KUKA KRL program: MyProgram_192().src

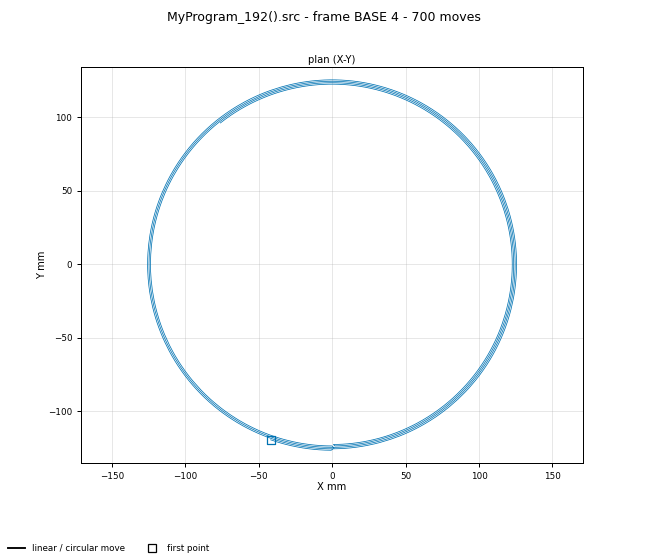
[picture p0: tool path of MyProgram_192().src in frame BASE 4, 700 of 700 moves have a stored position in this frame; points joined in program order, loops and branches not executed]
&ACCESS RVP
&REL 1
&PARAM TEMPLATE = C:\KRC\Roboter\Template\vorgabe
&PARAM EDITMASK = *
DEF MyProgram_192()
; ---- Setting reference (Base) ----
$BASE = BASE_DATA[4]

; --------------------------
; ---- Setting tool (TCP) ----
$TOOL = TOOL_DATA[3]
; --------------------------

$VEL.CP = VEL_APROX_PRINT
Startdeposition()
$VEL.CP = VEL_PRINT
LIN {X -41.8046,Y -119.4809,Z 139,A -112.1898,B 24.9633,C -1.4001,E1 24.9485,E2 558.5305} C_DIS
LIN {X -38.0832,Y -120.719,Z 139,A -110.4755,B 24.9635,C -1.3957,E1 24.953,E2 556.8235} C_DIS
LIN {X -35.043,Y -121.6367,Z 139,A -109.0218,B 24.9635,C -1.3954,E1 24.9569,E2 555.368} C_DIS
LIN {X -31.8921,Y -122.5017,Z 139,A -107.3287,B 24.963,C -1.405,E1 24.9616,E2 553.6497} C_DIS
LIN {X -27.5144,Y -123.5583,Z 139,A -105.3425,B 24.9632,C -1.4014,E1 24.967,E2 551.6695} C_DIS
LIN {X -23.703,Y -124.3439,Z 139,A -103.7035,B 24.9636,C -1.3947,E1 24.9714,E2 550.0445} C_DIS
LIN {X -20.2277,Y -124.9578,Z 139,A -102.0069,B 24.9633,C -1.399,E1 24.9761,E2 548.336} C_DIS
LIN {X -16.3797,Y -125.5188,Z 139,A -100.3777,B 24.9637,C -1.3922,E1 24.9806,E2 546.7217} C_DIS
LIN {X -12.7728,Y -125.9388,Z 139,A -98.5892,B 24.9633,C -1.3991,E1 24.9856,E2 544.9157} C_DIS
LIN {X -8.9623,Y -126.2657,Z 139,A -96.8687,B 24.9633,C -1.3986,E1 24.9904,E2 543.1957} C_DIS
LIN {X -4.8152,Y -126.4916,Z 139,A -95.0556,B 24.9635,C -1.3954,E1 24.9954,E2 541.3897} C_DIS
LIN {X -0.6506,Y -126.5815,Z 139,A -93.2386,B 24.9637,C -1.3924,E1 25.0005,E2 539.5799} C_DIS
LIN {X -0.6506,Y -126.5815,Z 139,A -93.2386,B 24.9637,C -1.3924,E1 25.0005,E2 539.5799} C_DIS
Enddeposition()
LIN {X 0.8997,Y -125.5994,Z 139,A -93.1322,B 24.9643,C -1.3803,E1 25.0007,E2 539.5021} C_DIS
Startdeposition()
$VEL.CP = VEL_PRINT
LIN {X -2.5774,Y -125.5787,Z 139,A -94.9255,B 24.9649,C -1.3699,E1 24.9956,E2 541.3201} C_DIS
LIN {X -6.6331,Y -125.4293,Z 139,A -96.7717,B 24.9649,C -1.3699,E1 24.9905,E2 543.1665} C_DIS
LIN {X -10.6993,Y -125.1476,Z 139,A -98.5659,B 24.9647,C -1.3732,E1 24.9855,E2 544.9538} C_DIS
LIN {X -14.9192,Y -124.7148,Z 139,A -100.4884,B 24.9647,C -1.374,E1 24.9802,E2 546.8756} C_DIS
LIN {X -18.8934,Y -124.1753,Z 139,A -102.3022,B 24.9646,C -1.3752,E1 24.9752,E2 548.688} C_DIS
LIN {X -22.2036,Y -123.6258,Z 139,A -103.8436,B 24.9646,C -1.3752,E1 24.9709,E2 550.2309} C_DIS
LIN {X -25.9892,Y -122.8868,Z 139,A -105.6556,B 24.9646,C -1.3734,E1 24.9659,E2 552.0493} C_DIS
LIN {X -28.9108,Y -122.2325,Z 139,A -107.185,B 24.965,C -1.3663,E1 24.9617,E2 553.5976} C_DIS
LIN {X -33.6478,Y -121.0131,Z 139,A -109.19,B 24.9644,C -1.3785,E1 24.9564,E2 555.5766} C_DIS
LIN {X -36.8186,Y -120.0862,Z 139,A -110.6976,B 24.9644,C -1.3796,E1 24.9523,E2 557.0842} C_DIS
LIN {X -39.7861,Y -119.1359,Z 139,A -112.2561,B 24.9646,C -1.3742,E1 24.9482,E2 558.6584} C_DIS
LIN {X -43.8401,Y -117.7047,Z 139,A -114.0437,B 24.9641,C -1.3842,E1 24.9435,E2 560.4258} C_DIS
LIN {X -46.4102,Y -116.7164,Z 139,A -115.4613,B 24.9644,C -1.3778,E1 24.9398,E2 561.8618} C_DIS
LIN {X -50.5279,Y -114.9946,Z 139,A -117.4765,B 24.9643,C -1.3809,E1 24.9346,E2 563.8741} C_DIS
LIN {X -53.8675,Y -113.4665,Z 139,A -119.0475,B 24.9639,C -1.3878,E1 24.9307,E2 565.4326} C_DIS
LIN {X -57.4932,Y -111.6742,Z 139,A -120.8939,B 24.9639,C -1.3901,E1 24.9261,E2 567.2786} C_DIS
LIN {X -60.8547,Y -109.8792,Z 139,A -122.6643,B 24.9638,C -1.391,E1 24.9217,E2 569.0519} C_DIS
LIN {X -64.9208,Y -107.5265,Z 139,A -125.2363,B 24.9646,C -1.3741,E1 24.9154,E2 571.6717} C_DIS
LIN {X -68.1564,Y -105.506,Z 139,A -126.6649,B 24.9637,C -1.3913,E1 24.9122,E2 573.0641} C_DIS
LIN {X -71.0171,Y -103.6017,Z 139,A -128.2398,B 24.9637,C -1.3936,E1 24.9085,E2 574.6388} C_DIS
LIN {X -74.697,Y -100.9815,Z 139,A -130.2962,B 24.9634,C -1.3974,E1 24.9039,E2 576.6934} C_DIS
LIN {X -77.4345,Y -98.8973,Z 139,A -132.2032,B 24.9641,C -1.3847,E1 24.8996,E2 578.6376} C_DIS
LIN {X -80.408,Y -96.4958,Z 139,A -133.6399,B 24.9632,C -1.4021,E1 24.8966,E2 580.0383} C_DIS
LIN {X -83.6363,Y -93.711,Z 139,A -135.5875,B 24.963,C -1.4059,E1 24.8925,E2 581.9846} C_DIS
LIN {X -86.9695,Y -90.6262,Z 139,A -137.6592,B 24.9627,C -1.4102,E1 24.8883,E2 584.0545} C_DIS
LIN {X -90.0345,Y -87.582,Z 139,A -139.6608,B 24.9626,C -1.4131,E1 24.8843,E2 586.0578} C_DIS
LIN {X -92.6006,Y -84.864,Z 139,A -141.6419,B 24.9631,C -1.4044,E1 24.8805,E2 588.0684} C_DIS
LIN {X -95.0006,Y -82.1687,Z 139,A -143.0168,B 24.9622,C -1.4205,E1 24.8781,E2 589.411} C_DIS
LIN {X -97.863,Y -78.7375,Z 139,A -144.9662,B 24.9617,C -1.4295,E1 24.8746,E2 591.3482} C_DIS
LIN {X -100.4945,Y -75.3509,Z 139,A -147.0461,B 24.9617,C -1.4287,E1 24.8711,E2 593.4399} C_DIS
LIN {X -102.9709,Y -71.929,Z 139,A -149.1222,B 24.9619,C -1.4269,E1 24.8677,E2 595.5306} C_DIS
LIN {X -105.0542,Y -68.8508,Z 139,A -150.9071,B 24.9619,C -1.4272,E1 24.865,E2 597.3235} C_DIS
LIN {X -106.8737,Y -65.9915,Z 139,A -152.244,B 24.9611,C -1.4408,E1 24.863,E2 598.6349} C_DIS
LIN {X -109.1521,Y -62.1496,Z 139,A -154.2487,B 24.9607,C -1.4478,E1 24.8602,E2 600.6332} C_DIS
LIN {X -110.9704,Y -58.8396,Z 139,A -155.9668,B 24.9605,C -1.4529,E1 24.858,E2 602.3485} C_DIS
LIN {X -113.9832,Y -52.7646,Z 139,A -159.0137,B 24.9599,C -1.4638,E1 24.8543,E2 605.3858} C_DIS
LIN {X -115.3845,Y -49.626,Z 139,A -160.6837,B 24.9599,C -1.4638,E1 24.8524,E2 607.065} C_DIS
LIN {X -116.9285,Y -45.8711,Z 139,A -162.312,B 24.959,C -1.4793,E1 24.8507,E2 608.6654} C_DIS
LIN {X -118.071,Y -42.844,Z 139,A -163.9544,B 24.9592,C -1.4763,E1 24.8491,E2 610.3244} C_DIS
LIN {X -119.1423,Y -39.7671,Z 139,A -165.4335,B 24.9589,C -1.4811,E1 24.8477,E2 611.8003} C_DIS
LIN {X -120.1236,Y -36.6965,Z 139,A -166.9045,B 24.9587,C -1.4856,E1 24.8465,E2 613.2691} C_DIS
LIN {X -121.1356,Y -33.2072,Z 139,A -168.7783,B 24.9589,C -1.481,E1 24.8451,E2 615.1646} C_DIS
LIN {X -122.133,Y -29.3235,Z 139,A -170.7253,B 24.9589,C -1.4815,E1 24.8438,E2 617.1219} C_DIS
LIN {X -123.4003,Y -23.4251,Z 139,A -172.8757,B 24.9569,C -1.5171,E1 24.8426,E2 619.2} C_DIS
LIN {X -124.2205,Y -18.6016,Z 139,A -175.544,B 24.9576,C -1.5047,E1 24.8414,E2 621.9139} C_DIS
LIN {X -124.7295,Y -14.7961,Z 139,A -177.2038,B 24.957,C -1.5145,E1 24.8408,E2 623.5604} C_DIS
LIN {X -125.2275,Y -9.7372,Z 139,A -179.7895,B 24.9573,C -1.5101,E1 24.8401,E2 626.1719} C_DIS
LIN {X -125.5171,Y -4.6805,Z 139,A 178.1039,B 24.9563,C -1.5267,E1 24.8399,E2 628.2515} C_DIS
LIN {X -125.5893,Y -1.9388,Z 139,A 176.6889,B 24.9565,C -1.5236,E1 24.8398,E2 629.6827} C_DIS
LIN {X -125.5414,Y 4.0033,Z 139,A 174.0819,B 24.9557,C -1.537,E1 24.8399,E2 632.2733} C_DIS
LIN {X -125.3591,Y 7.8425,Z 139,A 172.3326,B 24.9554,C -1.543,E1 24.8402,E2 634.0188} C_DIS
LIN {X -124.8359,Y 13.8763,Z 139,A 169.6269,B 24.9547,C -1.5546,E1 24.8409,E2 636.7132} C_DIS
LIN {X -124.0149,Y 19.9294,Z 139,A 166.6755,B 24.9547,C -1.5564,E1 24.8421,E2 639.6779} C_DIS
LIN {X -123.367,Y 23.5991,Z 139,A 165.0734,B 24.954,C -1.5663,E1 24.8429,E2 641.2658} C_DIS
LIN {X -122.5721,Y 27.4356,Z 139,A 163.0882,B 24.9542,C -1.5633,E1 24.844,E2 643.2698} C_DIS
LIN {X -121.449,Y 32.0403,Z 139,A 161.0453,B 24.9535,C -1.5756,E1 24.8454,E2 645.2954} C_DIS
LIN {X -120.3646,Y 35.9036,Z 139,A 159.278,B 24.953,C -1.5843,E1 24.8468,E2 647.0523} C_DIS
LIN {X -119.2699,Y 39.3837,Z 139,A 157.5521,B 24.9528,C -1.5868,E1 24.8483,E2 648.7819} C_DIS
LIN {X -118.0874,Y 42.7983,Z 139,A 155.8874,B 24.9526,C -1.5913,E1 24.8498,E2 650.4453} C_DIS
LIN {X -117.06,Y 45.5329,Z 139,A 154.2556,B 24.9531,C -1.5822,E1 24.8515,E2 652.108} C_DIS
LIN {X -115.836,Y 48.5627,Z 139,A 153.0432,B 24.9521,C -1.5992,E1 24.8527,E2 653.2867} C_DIS
LIN {X -113.2763,Y 54.2656,Z 139,A 150.184,B 24.9516,C -1.6076,E1 24.8561,E2 656.1415} C_DIS
LIN {X -111.744,Y 57.356,Z 139,A 148.3559,B 24.952,C -1.601,E1 24.8584,E2 657.9951} C_DIS
LIN {X -109.8749,Y 60.8626,Z 139,A 146.0208,B 24.953,C -1.5833,E1 24.8617,E2 660.3848} C_DIS
LIN {X -107.1204,Y 65.5894,Z 139,A 144.2085,B 24.9508,C -1.6208,E1 24.8641,E2 662.117} C_DIS
LIN {X -104.7423,Y 69.3244,Z 139,A 142.1709,B 24.9505,C -1.6258,E1 24.8672,E2 664.153} C_DIS
LIN {X -102.4969,Y 72.603,Z 139,A 140.3858,B 24.9501,C -1.6321,E1 24.8701,E2 665.9319} C_DIS
LIN {X -100.006,Y 75.9979,Z 139,A 138.3651,B 24.9501,C -1.6329,E1 24.8735,E2 667.9603} C_DIS
LIN {X -97.3017,Y 79.43,Z 139,A 136.4034,B 24.9496,C -1.6397,E1 24.8769,E2 669.9151} C_DIS
LIN {X -94.3922,Y 82.8673,Z 139,A 134.2991,B 24.9494,C -1.6428,E1 24.8807,E2 672.0215} C_DIS
LIN {X -91.6174,Y 85.9251,Z 139,A 132.405,B 24.9492,C -1.6471,E1 24.8843,E2 673.9137} C_DIS
LIN {X -88.5694,Y 89.0629,Z 139,A 130.4421,B 24.9488,C -1.6535,E1 24.8881,E2 675.8697} C_DIS
LIN {X -85.3469,Y 92.1562,Z 139,A 128.3653,B 24.9486,C -1.6566,E1 24.8924,E2 677.9476} C_DIS
LIN {X -82.2121,Y 94.9632,Z 139,A 126.4267,B 24.9483,C -1.6602,E1 24.8964,E2 679.8854} C_DIS
LIN {X -78.6759,Y 97.9126,Z 139,A 124.372,B 24.9479,C -1.667,E1 24.9008,E2 681.9317} C_DIS
LIN {X -75.5113,Y 100.3734,Z 139,A 122.5578,B 24.9476,C -1.6716,E1 24.9048,E2 683.7416} C_DIS
LIN {X -72.0749,Y 102.8694,Z 139,A 120.5324,B 24.9476,C -1.6716,E1 24.9095,E2 685.774} C_DIS
LIN {X -68.4195,Y 105.3352,Z 139,A 118.5413,B 24.9473,C -1.6765,E1 24.9141,E2 687.7599} C_DIS
LIN {X -64.6224,Y 107.7071,Z 139,A 115.7068,B 24.9493,C -1.6444,E1 24.9211,E2 690.6795} C_DIS
LIN {X -59.4468,Y 110.6473,Z 139,A 113.7306,B 24.9469,C -1.6827,E1 24.9257,E2 692.5704} C_DIS
LIN {X -55.8231,Y 112.5172,Z 139,A 112.2269,B 24.9457,C -1.7022,E1 24.9293,E2 694.0317} C_DIS
LIN {X -52.1716,Y 114.2574,Z 139,A 109.967,B 24.9467,C -1.6859,E1 24.9352,E2 696.3359} C_DIS
LIN {X -48.6833,Y 115.7856,Z 139,A 108.4077,B 24.9461,C -1.6967,E1 24.9391,E2 697.8732} C_DIS
LIN {X -45.6353,Y 117.0202,Z 139,A 106.8995,B 24.9459,C -1.6984,E1 24.943,E2 699.3806} C_DIS
LIN {X -41.9744,Y 118.3845,Z 139,A 103.8529,B 24.9494,C -1.6428,E1 24.9515,E2 702.5654} C_DIS
LIN {X -34.5296,Y 120.7665,Z 139,A 100.6379,B 24.9482,C -1.6627,E1 24.9599,E2 705.7385} C_DIS
LIN {X -28.6672,Y 122.2908,Z 139,A 98.159,B 24.9472,C -1.6783,E1 24.9666,E2 708.1834} C_DIS
LIN {X -24.1576,Y 123.2602,Z 139,A 96.5853,B 24.9455,C -1.7048,E1 24.9707,E2 709.6962} C_DIS
LIN {X -20.4182,Y 123.9335,Z 139,A 94.906,B 24.9453,C -1.7086,E1 24.9753,E2 711.3681} C_DIS
LIN {X -16.5856,Y 124.5044,Z 139,A 93.1652,B 24.9451,C -1.711,E1 24.9801,E2 713.1045} C_DIS
LIN {X -13.4064,Y 124.8865,Z 139,A 91.6264,B 24.9453,C -1.7082,E1 24.9844,E2 714.651} C_DIS
LIN {X -9.281,Y 125.2608,Z 139,A 89.7847,B 24.9451,C -1.7113,E1 24.9895,E2 716.4861} C_DIS
LIN {X -5.3106,Y 125.4925,Z 139,A 87.933,B 24.9451,C -1.7102,E1 24.9947,E2 718.3411} C_DIS
LIN {X -1.4943,Y 125.5967,Z 139,A 86.1631,B 24.9452,C -1.7093,E1 24.9996,E2 720.1132} C_DIS
LIN {X 2.1011,Y 125.5866,Z 139,A 84.5803,B 24.9451,C -1.7123,E1 25.004,E2 721.6887} C_DIS
LIN {X 6.1932,Y 125.4514,Z 139,A 82.7367,B 24.945,C -1.7136,E1 25.0092,E2 723.5288} C_DIS
LIN {X 9.8797,Y 125.2168,Z 139,A 80.918,B 24.9454,C -1.7071,E1 25.0143,E2 725.362} C_DIS
LIN {X 13.9908,Y 124.8236,Z 139,A 79.0735,B 24.9453,C -1.7087,E1 25.0194,E2 727.2014} C_DIS
LIN {X 17.7134,Y 124.3487,Z 139,A 77.4381,B 24.9451,C -1.712,E1 25.0239,E2 728.8277} C_DIS
LIN {X 21.5145,Y 123.7492,Z 139,A 75.65,B 24.9452,C -1.7098,E1 25.0288,E2 730.6192} C_DIS
LIN {X 25.5833,Y 122.9721,Z 139,A 73.4688,B 24.9462,C -1.6949,E1 25.0349,E2 732.8329} C_DIS
LIN {X 28.8679,Y 122.2428,Z 139,A 72.1891,B 24.9454,C -1.7063,E1 25.0383,E2 734.0838} C_DIS
LIN {X 32.3878,Y 121.3563,Z 139,A 70.5867,B 24.9454,C -1.7079,E1 25.0426,E2 735.6801} C_DIS
LIN {X 36.3536,Y 120.2285,Z 139,A 68.5283,B 24.946,C -1.6979,E1 25.0482,E2 737.7586} C_DIS
LIN {X 40.896,Y 118.7598,Z 139,A 66.5494,B 24.9455,C -1.7057,E1 25.0533,E2 739.7152} C_DIS
LIN {X 45.1754,Y 117.199,Z 139,A 64.4528,B 24.9457,C -1.7028,E1 25.0588,E2 741.8142} C_DIS
LIN {X 48.4633,Y 115.8775,Z 139,A 62.9005,B 24.9456,C -1.7042,E1 25.0628,E2 743.3596} C_DIS
LIN {X 51.3868,Y 114.611,Z 139,A 61.4504,B 24.9456,C -1.7027,E1 25.0665,E2 744.8097} C_DIS
LIN {X 54.4859,Y 113.1711,Z 139,A 59.5276,B 24.9469,C -1.683,E1 25.0715,E2 746.7742} C_DIS
LIN {X 57.6312,Y 111.6038,Z 139,A 58.3046,B 24.9459,C -1.6995,E1 25.0744,E2 747.9549} C_DIS
LIN {X 60.2766,Y 110.1975,Z 139,A 56.2801,B 24.948,C -1.6653,E1 25.0796,E2 750.0543} C_DIS
LIN {X 64.4594,Y 107.8042,Z 139,A 54.6424,B 24.9465,C -1.6895,E1 25.0834,E2 751.6298} C_DIS
LIN {X 68.1071,Y 105.5381,Z 139,A 52.6395,B 24.9468,C -1.6842,E1 25.0881,E2 753.6387} C_DIS
LIN {X 71.9524,Y 102.9547,Z 139,A 50.5794,B 24.9469,C -1.6833,E1 25.0928,E2 755.694} C_DIS
LIN {X 75.4343,Y 100.4315,Z 139,A 48.6447,B 24.947,C -1.6811,E1 25.0972,E2 757.627} C_DIS
LIN {X 79.735,Y 97.0517,Z 139,A 46.049,B 24.9477,C -1.6714,E1 25.1029,E2 760.2359} C_DIS
LIN {X 83.6029,Y 93.7409,Z 139,A 43.8076,B 24.9477,C -1.6707,E1 25.1076,E2 762.47} C_DIS
LIN {X 86.9996,Y 90.5972,Z 139,A 41.7098,B 24.9479,C -1.667,E1 25.1118,E2 764.5681} C_DIS
LIN {X 90.044,Y 87.5722,Z 139,A 39.7496,B 24.9482,C -1.6625,E1 25.1157,E2 766.5303} C_DIS
LIN {X 92.3902,Y 85.0928,Z 139,A 38.3722,B 24.9479,C -1.6681,E1 25.1183,E2 767.8887} C_DIS
LIN {X 94.875,Y 82.314,Z 139,A 36.5164,B 24.9486,C -1.6563,E1 25.1217,E2 769.764} C_DIS
LIN {X 97.6304,Y 79.0258,Z 139,A 34.5782,B 24.9488,C -1.6525,E1 25.1252,E2 771.7022} C_DIS
LIN {X 100.3697,Y 75.5162,Z 139,A 32.5251,B 24.9492,C -1.6463,E1 25.1287,E2 773.7601} C_DIS
LIN {X 102.808,Y 72.1619,Z 139,A 30.6579,B 24.9494,C -1.6427,E1 25.1317,E2 775.6267} C_DIS
LIN {X 105.2436,Y 68.5606,Z 139,A 28.7003,B 24.9497,C -1.6388,E1 25.1347,E2 777.5837} C_DIS
LIN {X 107.643,Y 64.7288,Z 139,A 26.9349,B 24.9491,C -1.6484,E1 25.1373,E2 779.3177} C_DIS
LIN {X 109.422,Y 61.6733,Z 139,A 25.0482,B 24.9502,C -1.63,E1 25.1399,E2 781.2379} C_DIS
LIN {X 111.6062,Y 57.6225,Z 139,A 22.4385,B 24.9521,C -1.5982,E1 25.1434,E2 783.9088} C_DIS
LIN {X 113.7419,Y 53.2865,Z 139,A 20.7741,B 24.9509,C -1.6193,E1 25.1453,E2 785.5145} C_DIS
LIN {X 115.2836,Y 49.8595,Z 139,A 19.1857,B 24.9508,C -1.6207,E1 25.1471,E2 787.0909} C_DIS
LIN {X 116.5335,Y 46.8639,Z 139,A 17.7529,B 24.9508,C -1.6188,E1 25.1486,E2 788.5204} C_DIS
LIN {X 117.6624,Y 43.9529,Z 139,A 16.2668,B 24.9513,C -1.6114,E1 25.1501,E2 790.0158} C_DIS
LIN {X 119.789,Y 37.7772,Z 139,A 13.5675,B 24.951,C -1.6167,E1 25.1525,E2 792.6873} C_DIS
LIN {X 121.2092,Y 32.9393,Z 139,A 10.9939,B 24.9523,C -1.5954,E1 25.1545,E2 795.2963} C_DIS
LIN {X 122.115,Y 29.398,Z 139,A 9.039,B 24.9535,C -1.5754,E1 25.1558,E2 797.2871} C_DIS
LIN {X 122.8724,Y 26.0559,Z 139,A 7.7703,B 24.9529,C -1.5855,E1 25.1566,E2 798.5245} C_DIS
LIN {X 123.6152,Y 22.2629,Z 139,A 6.0298,B 24.9532,C -1.5811,E1 25.1575,E2 800.2653} C_DIS
LIN {X 124.2666,Y 18.2882,Z 139,A 4.1797,B 24.9536,C -1.5745,E1 25.1583,E2 802.12} C_DIS
LIN {X 124.7327,Y 14.7691,Z 139,A 2.6323,B 24.9536,C -1.573,E1 25.1588,E2 803.6619} C_DIS
LIN {X 125.1456,Y 10.7228,Z 139,A 0.7912,B 24.954,C -1.5677,E1 25.1593,E2 805.5045} C_DIS
LIN {X 125.4112,Y 6.9924,Z 139,A -1.0044,B 24.9546,C -1.5574,E1 25.1596,E2 807.3136} C_DIS
LIN {X 125.5653,Y 3.1414,Z 139,A -2.6651,B 24.9546,C -1.5567,E1 25.1598,E2 808.9662} C_DIS
LIN {X 125.6025,Y -0.7041,Z 139,A -4.4232,B 24.9549,C -1.5508,E1 25.1598,E2 810.7279} C_DIS
LIN {X 125.5084,Y -4.9039,Z 139,A -6.3178,B 24.9552,C -1.5456,E1 25.1596,E2 812.6234} C_DIS
LIN {X 125.28,Y -9.018,Z 139,A -8.197,B 24.9556,C -1.5394,E1 25.1593,E2 814.5059} C_DIS
LIN {X 124.9403,Y -12.9066,Z 139,A -9.9541,B 24.9559,C -1.5347,E1 25.1588,E2 816.2637} C_DIS
LIN {X 124.5518,Y -16.2243,Z 139,A -11.4431,B 24.9561,C -1.5315,E1 25.1583,E2 817.7514} C_DIS
LIN {X 123.9986,Y -20.0282,Z 139,A -13.2581,B 24.9566,C -1.5226,E1 25.1575,E2 819.5769} C_DIS
LIN {X 123.4086,Y -23.3815,Z 139,A -14.6965,B 24.9566,C -1.5234,E1 25.1568,E2 821.0049} C_DIS
LIN {X 121.8269,Y -30.5719,Z 139,A -18.0743,B 24.9572,C -1.5115,E1 25.1547,E2 824.3912} C_DIS
LIN {X 120.8473,Y -34.2409,Z 139,A -20.0519,B 24.9582,C -1.4932,E1 25.1532,E2 826.4005} C_DIS
LIN {X 119.3517,Y -39.1383,Z 139,A -22.0859,B 24.9578,C -1.5013,E1 25.1516,E2 828.4039} C_DIS
LIN {X 117.7927,Y -43.605,Z 139,A -24.2456,B 24.9582,C -1.4943,E1 25.1495,E2 830.5679} C_DIS
LIN {X 116.5292,Y -46.8746,Z 139,A -26.2206,B 24.9595,C -1.47,E1 25.1474,E2 832.5893} C_DIS
LIN {X 115.1052,Y -50.2722,Z 139,A -27.5204,B 24.9587,C -1.4843,E1 25.1461,E2 833.8482} C_DIS
LIN {X 113.3225,Y -54.1691,Z 139,A -29.5136,B 24.9592,C -1.4763,E1 25.1437,E2 835.8495} C_DIS
LIN {X 111.3795,Y -58.0604,Z 139,A -31.4306,B 24.9593,C -1.4738,E1 25.1413,E2 837.7624} C_DIS
LIN {X 109.7344,Y -61.1163,Z 139,A -33.049,B 24.9597,C -1.4672,E1 25.1391,E2 839.3878} C_DIS
LIN {X 107.6373,Y -64.7383,Z 139,A -34.9579,B 24.96,C -1.4616,E1 25.1364,E2 841.3001} C_DIS
LIN {X 105.4653,Y -68.2191,Z 139,A -36.8491,B 24.9603,C -1.4551,E1 25.1335,E2 843.197} C_DIS
LIN {X 103.1553,Y -71.6641,Z 139,A -38.7026,B 24.9605,C -1.4517,E1 25.1306,E2 845.0494} C_DIS
LIN {X 100.6382,Y -75.1579,Z 139,A -41.1904,B 24.9623,C -1.4195,E1 25.1264,E2 847.6011} C_DIS
LIN {X 97.7463,Y -78.8822,Z 139,A -42.5715,B 24.9605,C -1.453,E1 25.1241,E2 848.8969} C_DIS
LIN {X 93.386,Y -83.9992,Z 139,A -46.2121,B 24.9625,C -1.4156,E1 25.1173,E2 852.6094} C_DIS
LIN {X 90.744,Y -86.8461,Z 139,A -47.7215,B 24.962,C -1.4244,E1 25.1145,E2 854.0913} C_DIS
LIN {X 85.6075,Y -91.9135,Z 139,A -50.8034,B 24.9619,C -1.427,E1 25.1083,E2 857.1543} C_DIS
LIN {X 80.0109,Y -96.8246,Z 139,A -54.0155,B 24.9618,C -1.4284,E1 25.1016,E2 860.3503} C_DIS
LIN {X 76.5271,Y -99.6013,Z 139,A -56.3022,B 24.9627,C -1.411,E1 25.0965,E2 862.6698} C_DIS
LIN {X 73.5795,Y -101.7979,Z 139,A -58.311,B 24.9638,C -1.3907,E1 25.0919,E2 864.7194} C_DIS
LIN {X 70.45,Y -103.9877,Z 139,A -59.6437,B 24.9629,C -1.4077,E1 25.0889,E2 866.0072} C_DIS
LIN {X 66.86,Y -106.3321,Z 139,A -61.6238,B 24.9631,C -1.4027,E1 25.0842,E2 867.993} C_DIS
LIN {X 63.4602,Y -108.3954,Z 139,A -63.4037,B 24.9632,C -1.401,E1 25.08,E2 869.7714} C_DIS
LIN {X 59.7756,Y -110.4706,Z 139,A -65.4413,B 24.9637,C -1.392,E1 25.075,E2 871.8241} C_DIS
LIN {X 55.8397,Y -112.509,Z 139,A -67.2931,B 24.9634,C -1.3972,E1 25.0704,E2 873.6587} C_DIS
LIN {X 52.8798,Y -113.9299,Z 139,A -68.765,B 24.9634,C -1.3961,E1 25.0667,E2 875.1294} C_DIS
LIN {X 49.8421,Y -115.2911,Z 139,A -70.3195,B 24.9637,C -1.3919,E1 25.0627,E2 876.6899} C_DIS
LIN {X 46.2319,Y -116.788,Z 139,A -72.1209,B 24.9639,C -1.3884,E1 25.058,E2 878.4956} C_DIS
LIN {X 39.8318,Y -119.1208,Z 139,A -75.2446,B 24.9641,C -1.3835,E1 25.0498,E2 881.6245} C_DIS
LIN {X 32.398,Y -121.3536,Z 139,A -78.6786,B 24.9641,C -1.3847,E1 25.0406,E2 885.0497} C_DIS
LIN {X 29.093,Y -122.1886,Z 139,A -80.3728,B 24.9645,C -1.3762,E1 25.036,E2 886.7615} C_DIS
LIN {X 23.7626,Y -123.3358,Z 139,A -82.7302,B 24.9643,C -1.3804,E1 25.0296,E2 889.106} C_DIS
LIN {X 20.4803,Y -123.9231,Z 139,A -84.2751,B 24.9644,C -1.378,E1 25.0253,E2 890.6549} C_DIS
LIN {X 16.4838,Y -124.5178,Z 139,A -86.1039,B 24.9644,C -1.3774,E1 25.0202,E2 892.4835} C_DIS
LIN {X 13.0103,Y -124.9291,Z 139,A -87.7746,B 24.9647,C -1.3728,E1 25.0156,E2 894.1641} C_DIS
LIN {X 9.2051,Y -125.2663,Z 139,A -89.4526,B 24.9646,C -1.3751,E1 25.0109,E2 895.8357} C_DIS
LIN {X 5.1896,Y -125.4972,Z 139,A -91.3048,B 24.9646,C -1.3735,E1 25.0058,E2 897.691} C_DIS
LIN {X 1.4055,Y -125.5982,Z 139,A -93.1062,B 24.9649,C -1.3693,E1 25.0007,E2 899.5021} C_DIS
LIN {X 1.4055,Y -125.5982,Z 139,A -93.1062,B 24.9649,C -1.3693,E1 25.0007,E2 899.5021} C_DIS
Enddeposition()
LIN {X 0.8898,Y -124.6193,Z 139,A -92.6917,B 24.7402,C -1.3712,E1 24.7777,E2 899.052} C_DIS
Startdeposition()
$VEL.CP = VEL_PRINT
LIN {X 4.2848,Y -124.5527,Z 139,A -90.8344,B 24.7394,C -1.386,E1 24.783,E2 897.1598} C_DIS
LIN {X 8.4379,Y -124.3407,Z 139,A -88.8956,B 24.7394,C -1.3881,E1 24.7884,E2 895.2167} C_DIS
LIN {X 12.3432,Y -124.013,Z 139,A -87.1688,B 24.7394,C -1.3855,E1 24.7932,E2 893.4973} C_DIS
LIN {X 16.3271,Y -123.5509,Z 139,A -85.358,B 24.7394,C -1.385,E1 24.7982,E2 891.689} C_DIS
LIN {X 20.3865,Y -122.9462,Z 139,A -83.4647,B 24.7394,C -1.3867,E1 24.8035,E2 889.7935} C_DIS
LIN {X 24.246,Y -122.2451,Z 139,A -81.4769,B 24.7388,C -1.3973,E1 24.809,E2 887.7827} C_DIS
LIN {X 29.506,Y -121.082,Z 139,A -79.1186,B 24.739,C -1.3939,E1 24.8154,E2 885.436} C_DIS
LIN {X 35.6088,Y -119.4306,Z 139,A -76.0112,B 24.7383,C -1.407,E1 24.8238,E2 882.3023} C_DIS
LIN {X 38.7371,Y -118.4534,Z 139,A -74.8992,B 24.7393,C -1.3893,E1 24.8266,E2 881.2349} C_DIS
LIN {X 43.968,Y -116.6113,Z 139,A -72.2971,B 24.7389,C -1.3952,E1 24.8335,E2 878.624} C_DIS
LIN {X 46.6782,Y -115.5528,Z 139,A -70.9573,B 24.7389,C -1.3973,E1 24.837,E2 877.2824} C_DIS
LIN {X 49.9084,Y -114.1958,Z 139,A -69.3718,B 24.7388,C -1.3984,E1 24.841,E2 875.6979} C_DIS
LIN {X 52.4782,Y -113.037,Z 139,A -68.0984,B 24.7388,C -1.3993,E1 24.8442,E2 874.4255} C_DIS
LIN {X 55.3568,Y -111.6556,Z 139,A -66.5505,B 24.7384,C -1.4057,E1 24.8482,E2 872.8665} C_DIS
LIN {X 59.3234,Y -109.6022,Z 139,A -64.4739,B 24.7381,C -1.4104,E1 24.8533,E2 870.7847} C_DIS
LIN {X 62.8966,Y -107.5911,Z 139,A -62.6268,B 24.7381,C -1.412,E1 24.8578,E2 868.9394} C_DIS
LIN {X 66.2174,Y -105.58,Z 139,A -60.7849,B 24.7377,C -1.4183,E1 24.8622,E2 867.0885} C_DIS
LIN {X 72.0177,Y -101.7117,Z 139,A -57.8149,B 24.738,C -1.4129,E1 24.869,E2 864.1414} C_DIS
LIN {X 74.5531,Y -99.868,Z 139,A -56.2235,B 24.7374,C -1.4235,E1 24.8726,E2 862.5304} C_DIS
LIN {X 77.7013,Y -97.4386,Z 139,A -54.1451,B 24.7365,C -1.4403,E1 24.8772,E2 860.42} C_DIS
LIN {X 83.0346,Y -92.9356,Z 139,A -51.315,B 24.7372,C -1.4284,E1 24.8831,E2 857.6293} C_DIS
LIN {X 85.688,Y -90.4952,Z 139,A -49.3607,B 24.7361,C -1.4475,E1 24.8872,E2 855.6376} C_DIS
LIN {X 89.1254,Y -87.1115,Z 139,A -46.8906,B 24.7351,C -1.466,E1 24.8921,E2 853.1342} C_DIS
LIN {X 91.999,Y -84.0718,Z 139,A -45.5115,B 24.7364,C -1.443,E1 24.8946,E2 851.8158} C_DIS
LIN {X 94.3596,Y -81.4127,Z 139,A -43.6973,B 24.7356,C -1.4565,E1 24.898,E2 849.9778} C_DIS
LIN {X 97.623,Y -77.4696,Z 139,A -41.1757,B 24.7348,C -1.4715,E1 24.9024,E2 847.4324} C_DIS
LIN {X 99.6902,Y -74.7913,Z 139,A -39.8815,B 24.7353,C -1.4624,E1 24.9046,E2 846.1662} C_DIS
LIN {X 102.1292,Y -71.4246,Z 139,A -37.9435,B 24.7349,C -1.4691,E1 24.9077,E2 844.2217} C_DIS
LIN {X 104.6692,Y -67.6474,Z 139,A -35.8911,B 24.7347,C -1.473,E1 24.9109,E2 842.1704} C_DIS
LIN {X 106.9158,Y -64.0378,Z 139,A -33.948,B 24.7344,C -1.4781,E1 24.9137,E2 840.225} C_DIS
LIN {X 109.1135,Y -60.2165,Z 139,A -31.9382,B 24.7341,C -1.4833,E1 24.9165,E2 838.2136} C_DIS
LIN {X 110.9573,Y -56.7434,Z 139,A -30.2376,B 24.7341,C -1.4833,E1 24.9186,E2 836.5221} C_DIS
LIN {X 112.4442,Y -53.7364,Z 139,A -28.6772,B 24.7338,C -1.4889,E1 24.9205,E2 834.9568} C_DIS
LIN {X 114.7458,Y -48.6318,Z 139,A -26.1521,B 24.7335,C -1.4943,E1 24.9234,E2 832.4328} C_DIS
LIN {X 116.34,Y -44.683,Z 139,A -24.0813,B 24.7328,C -1.5062,E1 24.9255,E2 830.3451} C_DIS
LIN {X 118.2353,Y -39.3922,Z 139,A -21.6094,B 24.7328,C -1.5087,E1 24.9278,E2 827.8815} C_DIS
LIN {X 120.3506,Y -32.3595,Z 139,A -18.3815,B 24.7325,C -1.5118,E1 24.9303,E2 824.6648} C_DIS
LIN {X 122.0316,Y -25.2955,Z 139,A -15.0989,B 24.7321,C -1.5197,E1 24.9324,E2 821.3827} C_DIS
LIN {X 122.5907,Y -22.4305,Z 139,A -13.5748,B 24.7313,C -1.5334,E1 24.9332,E2 819.835} C_DIS
LIN {X 123.1884,Y -18.8691,Z 139,A -11.9941,B 24.7313,C -1.5348,E1 24.9339,E2 818.2604} C_DIS
LIN {X 123.6997,Y -15.1637,Z 139,A -10.2299,B 24.7307,C -1.5427,E1 24.9345,E2 816.488} C_DIS
LIN {X 124.0871,Y -11.5717,Z 139,A -8.5663,B 24.7304,C -1.5483,E1 24.935,E2 814.8209} C_DIS
LIN {X 124.3946,Y -7.5762,Z 139,A -6.7813,B 24.7302,C -1.5514,E1 24.9353,E2 813.0393} C_DIS
LIN {X 124.5738,Y -3.5781,Z 139,A -4.9533,B 24.7299,C -1.5568,E1 24.9355,E2 811.2094} C_DIS
LIN {X 124.6251,Y 0.4016,Z 139,A -3.1032,B 24.7295,C -1.5639,E1 24.9355,E2 809.3537} C_DIS
LIN {X 124.5457,Y 4.4646,Z 139,A -1.2416,B 24.7291,C -1.5696,E1 24.9355,E2 807.4895} C_DIS
LIN {X 124.3419,Y 8.4219,Z 139,A 0.6319,B 24.7286,C -1.5782,E1 24.9351,E2 805.6069} C_DIS
LIN {X 124.0122,Y 12.3523,Z 139,A 2.3834,B 24.7285,C -1.5809,E1 24.9346,E2 803.8593} C_DIS
LIN {X 123.5552,Y 16.2944,Z 139,A 4.136,B 24.7283,C -1.5832,E1 24.934,E2 802.112} C_DIS
LIN {X 122.9787,Y 20.1921,Z 139,A 5.9495,B 24.728,C -1.5891,E1 24.9333,E2 800.2952} C_DIS
LIN {X 122.3673,Y 23.6145,Z 139,A 7.5213,B 24.7278,C -1.5928,E1 24.9325,E2 798.7238} C_DIS
LIN {X 121.3367,Y 28.442,Z 139,A 9.8571,B 24.7271,C -1.6034,E1 24.931,E2 796.3767} C_DIS
LIN {X 120.6478,Y 31.238,Z 139,A 11.3037,B 24.7265,C -1.6138,E1 24.93,E2 794.9137} C_DIS
LIN {X 118.6461,Y 38.1377,Z 139,A 14.7081,B 24.7255,C -1.6292,E1 24.9273,E2 791.4923} C_DIS
LIN {X 117.5304,Y 41.4531,Z 139,A 15.9204,B 24.7265,C -1.6137,E1 24.9262,E2 790.3236} C_DIS
LIN {X 116.3504,Y 44.6563,Z 139,A 17.6358,B 24.7257,C -1.6259,E1 24.9245,E2 788.5889} C_DIS
LIN {X 114.9929,Y 48.0409,Z 139,A 19.1975,B 24.7257,C -1.625,E1 24.9228,E2 787.038} C_DIS
LIN {X 113.6682,Y 51.0969,Z 139,A 20.7168,B 24.7256,C -1.6288,E1 24.9211,E2 785.518} C_DIS
LIN {X 110.8558,Y 56.9428,Z 139,A 23.5905,B 24.7254,C -1.6318,E1 24.9176,E2 782.6528} C_DIS
LIN {X 109.4961,Y 59.5181,Z 139,A 25.0729,B 24.7247,C -1.6428,E1 24.9156,E2 781.1521} C_DIS
LIN {X 106.9636,Y 63.9576,Z 139,A 27.1786,B 24.7251,C -1.6368,E1 24.9127,E2 779.0716} C_DIS
LIN {X 105.3162,Y 66.6353,Z 139,A 28.8462,B 24.7241,C -1.6519,E1 24.9102,E2 777.3766} C_DIS
LIN {X 103.0894,Y 70.0313,Z 139,A 30.7705,B 24.7236,C -1.6597,E1 24.9072,E2 775.4434} C_DIS
LIN {X 100.4559,Y 73.7589,Z 139,A 32.7751,B 24.7236,C -1.6603,E1 24.9039,E2 773.4472} C_DIS
LIN {X 97.8646,Y 77.1643,Z 139,A 34.7689,B 24.7232,C -1.6665,E1 24.9005,E2 771.4482} C_DIS
LIN {X 95.1545,Y 80.4827,Z 139,A 36.7098,B 24.723,C -1.6698,E1 24.897,E2 769.5085} C_DIS
LIN {X 92.3009,Y 83.7395,Z 139,A 38.4647,B 24.7235,C -1.6625,E1 24.8938,E2 767.7788} C_DIS
LIN {X 90.2609,Y 85.9347,Z 139,A 40.0734,B 24.7225,C -1.6772,E1 24.8907,E2 766.1423} C_DIS
LIN {X 87.2768,Y 88.9635,Z 139,A 42.1089,B 24.722,C -1.6855,E1 24.8867,E2 764.0957} C_DIS
LIN {X 83.9513,Y 92.1087,Z 139,A 44.1413,B 24.722,C -1.6863,E1 24.8825,E2 762.0699} C_DIS
LIN {X 80.5937,Y 95.0602,Z 139,A 46.538,B 24.7206,C -1.7074,E1 24.8773,E2 759.6322} C_DIS
LIN {X 77.5481,Y 97.5605,Z 139,A 47.7285,B 24.7224,C -1.6799,E1 24.8749,E2 758.5118} C_DIS
LIN {X 74.9635,Y 99.5603,Z 139,A 49.4822,B 24.7214,C -1.6951,E1 24.8709,E2 756.7283} C_DIS
LIN {X 71.4451,Y 102.1149,Z 139,A 51.385,B 24.7214,C -1.6938,E1 24.8666,E2 754.8353} C_DIS
LIN {X 68.1362,Y 104.3516,Z 139,A 53.1173,B 24.7216,C -1.6917,E1 24.8626,E2 753.1138} C_DIS
LIN {X 65.2751,Y 106.1647,Z 139,A 54.8376,B 24.7209,C -1.7022,E1 24.8585,E2 751.374} C_DIS
LIN {X 59.5496,Y 109.4789,Z 139,A 57.8885,B 24.7206,C -1.707,E1 24.8511,E2 748.3208} C_DIS
LIN {X 55.9103,Y 111.3814,Z 139,A 59.9611,B 24.7199,C -1.7186,E1 24.8459,E2 746.2264} C_DIS
LIN {X 52.0784,Y 113.2219,Z 139,A 61.5503,B 24.7209,C -1.7031,E1 24.842,E2 744.6783} C_DIS
LIN {X 49.4039,Y 114.414,Z 139,A 62.9817,B 24.7205,C -1.7088,E1 24.8383,E2 743.2368} C_DIS
LIN {X 46.111,Y 115.7815,Z 139,A 64.7281,B 24.7201,C -1.7157,E1 24.8337,E2 741.4779} C_DIS
LIN {X 42.4464,Y 117.1736,Z 139,A 66.3913,B 24.7204,C -1.7107,E1 24.8294,E2 739.8303} C_DIS
LIN {X 39.2901,Y 118.2693,Z 139,A 67.9053,B 24.7204,C -1.7109,E1 24.8254,E2 738.3186} C_DIS
LIN {X 36.2917,Y 119.2236,Z 139,A 69.3933,B 24.7202,C -1.7141,E1 24.8214,E2 736.8258} C_DIS
LIN {X 32.5438,Y 120.3015,Z 139,A 70.9943,B 24.7207,C -1.7061,E1 24.8172,E2 735.2467} C_DIS
LIN {X 27.0459,Y 121.6563,Z 139,A 73.9158,B 24.7196,C -1.7228,E1 24.8092,E2 732.2894} C_DIS
LIN {X 23.1348,Y 122.459,Z 139,A 75.5657,B 24.7201,C -1.7147,E1 24.8047,E2 730.6607} C_DIS
LIN {X 19.4654,Y 123.096,Z 139,A 77.3582,B 24.7198,C -1.7192,E1 24.7997,E2 728.8595} C_DIS
LIN {X 15.9457,Y 123.6009,Z 139,A 79.0222,B 24.7198,C -1.721,E1 24.7951,E2 727.1926} C_DIS
LIN {X 11.9288,Y 124.0528,Z 139,A 80.8105,B 24.7199,C -1.7179,E1 24.7902,E2 725.4128} C_DIS
LIN {X 7.8899,Y 124.3753,Z 139,A 82.6621,B 24.7199,C -1.7174,E1 24.785,E2 723.5632} C_DIS
LIN {X 4.35,Y 124.5502,Z 139,A 84.3557,B 24.7197,C -1.7204,E1 24.7803,E2 721.8631} C_DIS
LIN {X 0.5163,Y 124.6242,Z 139,A 86.0298,B 24.72,C -1.7159,E1 24.7756,E2 720.1998} C_DIS
LIN {X -3.1954,Y 124.5844,Z 139,A 87.7906,B 24.7199,C -1.7181,E1 24.7707,E2 718.4338} C_DIS
LIN {X -7.0576,Y 124.4266,Z 139,A 89.6347,B 24.7197,C -1.7206,E1 24.7656,E2 716.5833} C_DIS
LIN {X -10.8165,Y 124.1552,Z 139,A 91.3202,B 24.7199,C -1.7176,E1 24.7609,E2 714.9041} C_DIS
LIN {X -14.6607,Y 123.7597,Z 139,A 93.0627,B 24.7201,C -1.715,E1 24.7561,E2 713.1667} C_DIS
LIN {X -18.5212,Y 123.2422,Z 139,A 94.9162,B 24.72,C -1.7167,E1 24.7509,E2 711.3076} C_DIS
LIN {X -22.0847,Y 122.6526,Z 139,A 96.5309,B 24.7202,C -1.7134,E1 24.7465,E2 709.6993} C_DIS
LIN {X -28.1769,Y 121.3985,Z 139,A 99.6951,B 24.7194,C -1.725,E1 24.7378,E2 706.5032} C_DIS
LIN {X -31.4227,Y 120.6004,Z 139,A 100.8579,B 24.7207,C -1.7061,E1 24.7347,E2 705.3841} C_DIS
LIN {X -35.137,Y 119.569,Z 139,A 102.6964,B 24.7206,C -1.7073,E1 24.7298,E2 703.5398} C_DIS
LIN {X -42.2278,Y 117.2524,Z 139,A 106.1534,B 24.7208,C -1.7043,E1 24.7207,E2 700.0834} C_DIS
LIN {X -45.4976,Y 116.0233,Z 139,A 107.7439,B 24.721,C -1.7014,E1 24.7165,E2 698.4965} C_DIS
LIN {X -49.1747,Y 114.5131,Z 139,A 109.5947,B 24.721,C -1.6998,E1 24.7117,E2 696.6452} C_DIS
LIN {X -57.3599,Y 110.6416,Z 139,A 113.6707,B 24.7218,C -1.689,E1 24.7015,E2 692.5844} C_DIS
LIN {X -64.0611,Y 106.9019,Z 139,A 117.3112,B 24.7218,C -1.6878,E1 24.6927,E2 688.9361} C_DIS
LIN {X -67.5372,Y 104.7408,Z 139,A 119.3174,B 24.7218,C -1.6898,E1 24.6879,E2 686.9186} C_DIS
LIN {X -71.2956,Y 102.2189,Z 139,A 121.3502,B 24.7221,C -1.6835,E1 24.6832,E2 684.8941} C_DIS
LIN {X -74.7526,Y 99.7194,Z 139,A 123.3042,B 24.7224,C -1.679,E1 24.6788,E2 682.9437} C_DIS
LIN {X -77.9894,Y 97.2086,Z 139,A 125.2053,B 24.7226,C -1.6757,E1 24.6747,E2 681.0435} C_DIS
LIN {X -81.0592,Y 94.6641,Z 139,A 127.1099,B 24.7226,C -1.6748,E1 24.6706,E2 679.1337} C_DIS
LIN {X -84.4407,Y 91.6599,Z 139,A 129.1546,B 24.7231,C -1.6684,E1 24.6664,E2 677.0962} C_DIS
LIN {X -87.5869,Y 88.659,Z 139,A 131.2073,B 24.7232,C -1.6659,E1 24.6623,E2 675.0406} C_DIS
LIN {X -90.6143,Y 85.5617,Z 139,A 133.1431,B 24.7237,C -1.6585,E1 24.6585,E2 673.1143} C_DIS
LIN {X -93.5813,Y 82.3067,Z 139,A 135.2106,B 24.7239,C -1.6552,E1 24.6547,E2 671.0453} C_DIS
LIN {X -96.3175,Y 79.0871,Z 139,A 137.164,B 24.7242,C -1.6505,E1 24.6512,E2 669.094} C_DIS
LIN {X -98.9657,Y 75.7466,Z 139,A 139.1276,B 24.7245,C -1.6454,E1 24.6478,E2 667.1333} C_DIS
LIN {X -101.5185,Y 72.2898,Z 139,A 141.0678,B 24.725,C -1.6384,E1 24.6447,E2 665.2005} C_DIS
LIN {X -103.733,Y 69.0741,Z 139,A 142.8809,B 24.7252,C -1.6341,E1 24.6418,E2 663.3886} C_DIS
LIN {X -105.9537,Y 65.6174,Z 139,A 145.0994,B 24.7247,C -1.6434,E1 24.6385,E2 661.1363} C_DIS
LIN {X -107.7145,Y 62.6843,Z 139,A 146.465,B 24.7255,C -1.6295,E1 24.6366,E2 659.7969} C_DIS
LIN {X -109.4171,Y 59.6628,Z 139,A 147.968,B 24.7261,C -1.6207,E1 24.6346,E2 658.3071} C_DIS
LIN {X -111.0611,Y 56.5395,Z 139,A 149.5535,B 24.7265,C -1.6142,E1 24.6326,E2 656.7286} C_DIS
LIN {X -112.5319,Y 53.5529,Z 139,A 151.2487,B 24.7263,C -1.6169,E1 24.6305,E2 655.0177} C_DIS
LIN {X -114.2654,Y 49.7476,Z 139,A 152.8098,B 24.7276,C -1.595,E1 24.6288,E2 653.5006} C_DIS
LIN {X -115.6187,Y 46.5147,Z 139,A 154.6924,B 24.7272,C -1.602,E1 24.6267,E2 651.5907} C_DIS
LIN {X -116.8494,Y 43.3325,Z 139,A 156.3538,B 24.7272,C -1.6012,E1 24.6251,E2 649.9217} C_DIS
LIN {X -118.2372,Y 39.3862,Z 139,A 158.14,B 24.728,C -1.589,E1 24.6235,E2 648.1545} C_DIS
LIN {X -119.1981,Y 36.3753,Z 139,A 159.5943,B 24.7283,C -1.5845,E1 24.6223,E2 646.7027} C_DIS
LIN {X -120.1332,Y 33.1592,Z 139,A 161.267,B 24.7283,C -1.5854,E1 24.621,E2 645.0179} C_DIS
LIN {X -121.1591,Y 29.186,Z 139,A 163.0612,B 24.7288,C -1.5752,E1 24.6198,E2 643.2376} C_DIS
LIN {X -122.3335,Y 23.7916,Z 139,A 165.8375,B 24.7287,C -1.5775,E1 24.6182,E2 640.4393} C_DIS
LIN {X -123.7374,Y 14.8476,Z 139,A 169.5146,B 24.7308,C -1.5424,E1 24.6167,E2 636.8244} C_DIS
LIN {X -124.3122,Y 8.8285,Z 139,A 172.5271,B 24.7307,C -1.5434,E1 24.6159,E2 633.7912} C_DIS
LIN {X -124.4899,Y 5.8199,Z 139,A 174.6798,B 24.7289,C -1.573,E1 24.6156,E2 631.5543} C_DIS
LIN {X -124.6218,Y 0.99,Z 139,A 176.7161,B 24.7299,C -1.5574,E1 24.6156,E2 629.543} C_DIS
LIN {X -124.5922,Y -2.9176,Z 139,A 177.9475,B 24.7317,C -1.5264,E1 24.6156,E2 628.3787} C_DIS
LIN {X -124.4858,Y -5.9016,Z 139,A 179.9786,B 24.7302,C -1.5512,E1 24.6159,E2 626.2756} C_DIS
LIN {X -124.2152,Y -10.106,Z 139,A -178.0263,B 24.7305,C -1.5475,E1 24.6164,E2 624.2773} C_DIS
LIN {X -123.78,Y -14.4905,Z 139,A -176.6358,B 24.7325,C -1.5127,E1 24.6168,E2 622.9621} C_DIS
LIN {X -123.3705,Y -17.6381,Z 139,A -174.4665,B 24.7309,C -1.5397,E1 24.6177,E2 620.7149} C_DIS
LIN {X -122.6224,Y -22.2522,Z 139,A -172.9657,B 24.733,C -1.5038,E1 24.6184,E2 619.2913} C_DIS
LIN {X -121.3213,Y -28.5131,Z 139,A -169.9812,B 24.7334,C -1.4965,E1 24.6201,E2 616.3067} C_DIS
LIN {X -120.4879,Y -31.8445,Z 139,A -168.1594,B 24.7331,C -1.5024,E1 24.6214,E2 614.4599} C_DIS
LIN {X -119.117,Y -36.6403,Z 139,A -166.0383,B 24.7339,C -1.4877,E1 24.6231,E2 612.3619} C_DIS
LIN {X -117.8303,Y -40.5883,Z 139,A -164.1337,B 24.7342,C -1.4817,E1 24.6247,E2 610.4607} C_DIS
LIN {X -116.6921,Y -43.7523,Z 139,A -162.5268,B 24.7343,C -1.4798,E1 24.6263,E2 608.8491} C_DIS
LIN {X -115.5328,Y -46.7279,Z 139,A -161.1274,B 24.7348,C -1.4723,E1 24.6277,E2 607.4598} C_DIS
LIN {X -114.0894,Y -50.1547,Z 139,A -158.8776,B 24.7337,C -1.4916,E1 24.6303,E2 605.151} C_DIS
LIN {X -112.4186,Y -53.79,Z 139,A -157.4473,B 24.735,C -1.4679,E1 24.632,E2 603.7699} C_DIS
LIN {X -110.9581,Y -56.7418,Z 139,A -156.0147,B 24.7354,C -1.46,E1 24.6337,E2 602.3485} C_DIS
LIN {X -109.2505,Y -59.9682,Z 139,A -154.2264,B 24.7354,C -1.4602,E1 24.6361,E2 600.5501} C_DIS
LIN {X -107.1516,Y -63.6423,Z 139,A -152.2922,B 24.7357,C -1.4545,E1 24.6388,E2 598.6196} C_DIS
LIN {X -104.3608,Y -68.1225,Z 139,A -150.0883,B 24.7367,C -1.438,E1 24.6421,E2 596.444} C_DIS
LIN {X -102.2106,Y -71.3076,Z 139,A -148.1447,B 24.7365,C -1.4414,E1 24.6452,E2 594.4825} C_DIS
LIN {X -99.926,Y -74.4752,Z 139,A -146.2795,B 24.7365,C -1.44,E1 24.6483,E2 592.6114} C_DIS
LIN {X -97.2829,Y -77.8968,Z 139,A -144.415,B 24.7371,C -1.4296,E1 24.6515,E2 590.7631} C_DIS
LIN {X -95.186,Y -80.4457,Z 139,A -142.4484,B 24.7362,C -1.4465,E1 24.6551,E2 588.7468} C_DIS
LIN {X -92.9184,Y -83.0538,Z 139,A -141.1557,B 24.7371,C -1.4293,E1 24.6574,E2 587.4896} C_DIS
LIN {X -90.4486,Y -85.7373,Z 139,A -139.4633,B 24.7373,C -1.4262,E1 24.6606,E2 585.797} C_DIS
LIN {X -87.5,Y -88.7446,Z 139,A -137.4655,B 24.7373,C -1.4249,E1 24.6646,E2 583.7939} C_DIS
LIN {X -84.2463,Y -91.8386,Z 139,A -135.4801,B 24.7378,C -1.417,E1 24.6686,E2 581.8193} C_DIS
LIN {X -81.2183,Y -94.5271,Z 139,A -133.1772,B 24.7369,C -1.4337,E1 24.6736,E2 579.4672} C_DIS
LIN {X -78.1714,Y -97.0615,Z 139,A -131.7474,B 24.7381,C -1.4121,E1 24.6766,E2 578.0838} C_DIS
LIN {X -74.7573,Y -99.7159,Z 139,A -129.7006,B 24.7381,C -1.4112,E1 24.6811,E2 576.0317} C_DIS
LIN {X -71.2086,Y -102.2795,Z 139,A -127.8769,B 24.7387,C -1.399,E1 24.6852,E2 574.2308} C_DIS
LIN {X -68.3413,Y -104.2174,Z 139,A -126.1141,B 24.7385,C -1.4043,E1 24.6894,E2 572.4493} C_DIS
LIN {X -62.8207,Y -107.6357,Z 139,A -123.3214,B 24.7392,C -1.3908,E1 24.696,E2 569.6802} C_DIS
LIN {X -60.031,Y -109.216,Z 139,A -121.6146,B 24.7387,C -1.3996,E1 24.7002,E2 567.9473} C_DIS
LIN {X -55.8424,Y -111.416,Z 139,A -119.5797,B 24.7392,C -1.3902,E1 24.7052,E2 565.9293} C_DIS
LIN {X -51.7037,Y -113.3951,Z 139,A -117.3297,B 24.739,C -1.3944,E1 24.7109,E2 563.6637} C_DIS
LIN {X -47.2464,Y -115.3238,Z 139,A -115.2591,B 24.7395,C -1.3843,E1 24.7162,E2 561.6123} C_DIS
LIN {X -43.072,Y -116.9469,Z 139,A -112.9852,B 24.7391,C -1.3925,E1 24.7222,E2 559.3141} C_DIS
LIN {X -39.1952,Y -118.3009,Z 139,A -111.2385,B 24.7395,C -1.3843,E1 24.7268,E2 557.5837} C_DIS
LIN {X -36.1095,Y -119.2794,Z 139,A -109.8157,B 24.7397,C -1.38,E1 24.7306,E2 556.1685} C_DIS
LIN {X -32.8717,Y -120.2136,Z 139,A -107.923,B 24.7389,C -1.3953,E1 24.7358,E2 554.2362} C_DIS
LIN {X -27.8196,Y -121.4801,Z 139,A -105.7794,B 24.7396,C -1.3821,E1 24.7415,E2 552.1214} C_DIS
LIN {X -24.168,Y -122.261,Z 139,A -103.9627,B 24.7394,C -1.3861,E1 24.7465,E2 550.293} C_DIS
LIN {X -20.2719,Y -122.9654,Z 139,A -102.2689,B 24.7398,C -1.3795,E1 24.7511,E2 548.6134} C_DIS
LIN {X -16.385,Y -123.5433,Z 139,A -100.4505,B 24.7398,C -1.3795,E1 24.7562,E2 546.7932} C_DIS
LIN {X -13.1533,Y -123.9291,Z 139,A -98.9434,B 24.7398,C -1.3799,E1 24.7604,E2 545.2843} C_DIS
LIN {X -9.1507,Y -124.2887,Z 139,A -97.133,B 24.7398,C -1.378,E1 24.7654,E2 543.4776} C_DIS
LIN {X -5.5807,Y -124.5019,Z 139,A -95.3628,B 24.7395,C -1.3842,E1 24.7704,E2 541.6921} C_DIS
LIN {X -1.7199,Y -124.6138,Z 139,A -93.6351,B 24.7396,C -1.3822,E1 24.7752,E2 539.9692} C_DIS
LIN {X 0.8898,Y -124.6193,Z 139,A -92.6893,B 24.7403,C -1.3702,E1 24.7777,E2 539.052} C_DIS
Enddeposition()
LIN {X 0.8898,Y -124.6193,Z 139,A -92.6893,B 24.7403,C -1.3702,E1 24.7777,E2 539.052} C_DIS
Startdeposition()
$VEL.CP = VEL_PRINT
LIN {X -0.0893,Y -123.6476,Z 139,A -93.6074,B 24.2479,C -1.2635,E1 24.2776,E2 540.159} C_DIS
LIN {X -3.8094,Y -123.588,Z 139,A -95.347,B 24.2479,C -1.2625,E1 24.2728,E2 541.9012} C_DIS
LIN {X -7.7312,Y -123.4042,Z 139,A -97.1167,B 24.2478,C -1.2648,E1 24.2678,E2 543.6661} C_DIS
LIN {X -11.6102,Y -123.0999,Z 139,A -98.8989,B 24.2478,C -1.2658,E1 24.2629,E2 545.4466} C_DIS
LIN {X -15.6582,Y -122.6512,Z 139,A -100.8195,B 24.2478,C -1.2646,E1 24.2575,E2 547.3715} C_DIS
LIN {X -19.5403,Y -122.0938,Z 139,A -102.6819,B 24.2478,C -1.263,E1 24.2524,E2 549.2394} C_DIS
LIN {X -22.902,Y -121.5068,Z 139,A -104.1514,B 24.2476,C -1.2687,E1 24.2484,E2 550.6965} C_DIS
LIN {X -26.3434,Y -120.8072,Z 139,A -105.6997,B 24.2474,C -1.273,E1 24.2442,E2 552.2362} C_DIS
LIN {X -32.1873,Y -119.3833,Z 139,A -108.2712,B 24.2468,C -1.2844,E1 24.2373,E2 554.7836} C_DIS
LIN {X -35.4463,Y -118.4582,Z 139,A -110.2144,B 24.2476,C -1.2685,E1 24.2319,E2 556.769} C_DIS
LIN {X -38.8532,Y -117.3829,Z 139,A -111.8268,B 24.2475,C -1.2717,E1 24.2277,E2 558.3764} C_DIS
LIN {X -42.3003,Y -116.1856,Z 139,A -113.5933,B 24.2475,C -1.2698,E1 24.223,E2 560.1512} C_DIS
LIN {X -45.9469,Y -114.7921,Z 139,A -115.3422,B 24.2473,C -1.2743,E1 24.2185,E2 561.8931} C_DIS
LIN {X -49.5359,Y -113.2903,Z 139,A -117.2024,B 24.2473,C -1.2737,E1 24.2137,E2 563.7593} C_DIS
LIN {X -53.0459,Y -111.689,Z 139,A -118.7681,B 24.2468,C -1.2857,E1 24.2098,E2 565.2996} C_DIS
LIN {X -56.0581,Y -110.2076,Z 139,A -120.4608,B 24.247,C -1.2815,E1 24.2055,E2 567.0072} C_DIS
LIN {X -58.9331,Y -108.6999,Z 139,A -122.0852,B 24.2471,C -1.2781,E1 24.2015,E2 568.6445} C_DIS
LIN {X -62.7777,Y -106.5255,Z 139,A -123.8109,B 24.2463,C -1.2954,E1 24.1974,E2 570.3334} C_DIS
LIN {X -65.6395,Y -104.7869,Z 139,A -125.6679,B 24.2468,C -1.2841,E1 24.1929,E2 572.2239} C_DIS
LIN {X -69.069,Y -102.5585,Z 139,A -127.7131,B 24.247,C -1.2806,E1 24.1881,E2 574.2847} C_DIS
LIN {X -73.1153,Y -99.7139,Z 139,A -129.8488,B 24.2465,C -1.2914,E1 24.1833,E2 576.4016} C_DIS
LIN {X -75.9428,Y -97.5779,Z 139,A -132.3568,B 24.2482,C -1.2566,E1 24.1776,E2 579.0042} C_DIS
LIN {X -80.6332,Y -93.7389,Z 139,A -134.3703,B 24.2462,C -1.2966,E1 24.1735,E2 580.928} C_DIS
LIN {X -83.0852,Y -91.5726,Z 139,A -135.881,B 24.2461,C -1.2999,E1 24.1703,E2 582.4369} C_DIS
LIN {X -86.2727,Y -88.5767,Z 139,A -137.9427,B 24.2459,C -1.3026,E1 24.1662,E2 584.5008} C_DIS
LIN {X -89.2877,Y -85.5361,Z 139,A -139.8137,B 24.2454,C -1.3119,E1 24.1625,E2 586.3574} C_DIS
LIN {X -94.8662,Y -79.3041,Z 139,A -143.4907,B 24.2445,C -1.3293,E1 24.1558,E2 590.0087} C_DIS
LIN {X -97.1786,Y -76.4527,Z 139,A -145.4877,B 24.245,C -1.3206,E1 24.1522,E2 592.0367} C_DIS
LIN {X -99.8394,Y -72.9444,Z 139,A -147.5906,B 24.2449,C -1.3229,E1 24.1487,E2 594.1444} C_DIS
LIN {X -102.415,Y -69.281,Z 139,A -149.6705,B 24.2446,C -1.3281,E1 24.1454,E2 596.2224} C_DIS
LIN {X -104.3941,Y -66.262,Z 139,A -151.3498,B 24.2444,C -1.3321,E1 24.1429,E2 597.9004} C_DIS
LIN {X -106.6994,Y -62.4817,Z 139,A -153.38,B 24.2441,C -1.3386,E1 24.14,E2 599.9256} C_DIS
LIN {X -108.6548,Y -59.016,Z 139,A -155.2466,B 24.2439,C -1.3427,E1 24.1374,E2 601.7924} C_DIS
LIN {X -110.6351,Y -55.2125,Z 139,A -158.5239,B 24.2464,C -1.2938,E1 24.1332,E2 605.2076} C_DIS
LIN {X -114.0323,Y -47.8008,Z 139,A -160.7707,B 24.2425,C -1.3694,E1 24.1309,E2 607.2821} C_DIS
LIN {X -115.5735,Y -43.9476,Z 139,A -162.9838,B 24.2428,C -1.3626,E1 24.1286,E2 609.5246} C_DIS
LIN {X -116.8001,Y -40.5709,Z 139,A -164.5912,B 24.2424,C -1.3701,E1 24.1271,E2 611.1231} C_DIS
LIN {X -118.0311,Y -36.843,Z 139,A -166.52,B 24.2424,C -1.3709,E1 24.1255,E2 613.0613} C_DIS
LIN {X -119.2713,Y -32.6061,Z 139,A -168.472,B 24.2418,C -1.3812,E1 24.124,E2 614.9999} C_DIS
LIN {X -120.1209,Y -29.315,Z 139,A -170.0549,B 24.2416,C -1.3858,E1 24.1229,E2 616.5811} C_DIS
LIN {X -121.0136,Y -25.3869,Z 139,A -172.0861,B 24.2416,C -1.3846,E1 24.1217,E2 618.6275} C_DIS
LIN {X -122.3766,Y -17.6725,Z 139,A -175.4719,B 24.2405,C -1.4065,E1 24.1201,E2 621.9805} C_DIS
LIN {X -123.2015,Y -10.4753,Z 139,A -179.1119,B 24.2405,C -1.4053,E1 24.119,E2 625.646} C_DIS
LIN {X -123.5483,Y -4.9174,Z 139,A 178.6222,B 24.2393,C -1.4269,E1 24.1187,E2 627.8729} C_DIS
LIN {X -123.6409,Y 1.32,Z 139,A 175.3229,B 24.2398,C -1.419,E1 24.1187,E2 631.2121} C_DIS
LIN {X -123.4587,Y 6.8338,Z 139,A 173.0302,B 24.2387,C -1.4385,E1 24.1189,E2 633.4715} C_DIS
LIN {X -122.9142,Y 13.4345,Z 139,A 169.9906,B 24.2381,C -1.4497,E1 24.1196,E2 636.5024} C_DIS
LIN {X -122.2589,Y 18.474,Z 139,A 167.4129,B 24.2381,C -1.4479,E1 24.1206,E2 639.1004} C_DIS
LIN {X -121.6567,Y 22.092,Z 139,A 165.3321,B 24.2387,C -1.4375,E1 24.1216,E2 641.2197} C_DIS
LIN {X -120.9239,Y 25.803,Z 139,A 163.9562,B 24.2375,C -1.4589,E1 24.1224,E2 642.5513} C_DIS
LIN {X -120.0949,Y 29.423,Z 139,A 162.2889,B 24.2371,C -1.4667,E1 24.1234,E2 644.2097} C_DIS
LIN {X -119.1785,Y 32.9379,Z 139,A 160.5415,B 24.237,C -1.4694,E1 24.1247,E2 645.961} C_DIS
LIN {X -118.163,Y 36.4119,Z 139,A 158.8908,B 24.2366,C -1.4758,E1 24.126,E2 647.6058} C_DIS
LIN {X -116.9923,Y 40.0166,Z 139,A 157.0556,B 24.2365,C -1.478,E1 24.1276,E2 649.4464} C_DIS
LIN {X -115.6752,Y 43.6761,Z 139,A 154.6694,B 24.2375,C -1.4592,E1 24.13,E2 651.8927} C_DIS
LIN {X -113.9141,Y 48.0838,Z 139,A 153.1735,B 24.2355,C -1.4955,E1 24.1315,E2 653.3083} C_DIS
LIN {X -112.4128,Y 51.4955,Z 139,A 151.3535,B 24.2354,C -1.4968,E1 24.1336,E2 655.1353} C_DIS
LIN {X -110.9886,Y 54.4961,Z 139,A 149.8262,B 24.2351,C -1.502,E1 24.1355,E2 656.6586} C_DIS
LIN {X -109.5606,Y 57.3125,Z 139,A 148.4256,B 24.2347,C -1.509,E1 24.1372,E2 658.0497} C_DIS
LIN {X -107.8534,Y 60.4679,Z 139,A 146.6039,B 24.2347,C -1.5071,E1 24.1397,E2 659.8859} C_DIS
LIN {X -104.9154,Y 65.4329,Z 139,A 143.8888,B 24.2344,C -1.5131,E1 24.1436,E2 662.6009} C_DIS
LIN {X -102.7506,Y 68.7825,Z 139,A 142.0888,B 24.234,C -1.5203,E1 24.1464,E2 664.3925} C_DIS
LIN {X -100.3993,Y 72.1719,Z 139,A 140.1222,B 24.2338,C -1.5233,E1 24.1495,E2 666.3619} C_DIS
LIN {X -97.9304,Y 75.488,Z 139,A 138.1302,B 24.2338,C -1.5252,E1 24.1529,E2 668.359} C_DIS
LIN {X -95.0379,Y 79.0985,Z 139,A 136.0216,B 24.2333,C -1.5324,E1 24.1566,E2 670.4601} C_DIS
LIN {X -92.3196,Y 82.255,Z 139,A 134.0332,B 24.2331,C -1.5349,E1 24.1603,E2 672.4517} C_DIS
LIN {X -89.2502,Y 85.5753,Z 139,A 131.9633,B 24.2328,C -1.5412,E1 24.1642,E2 674.5155} C_DIS
LIN {X -86.2463,Y 88.6024,Z 139,A 129.9472,B 24.2326,C -1.5443,E1 24.1682,E2 676.5328} C_DIS
LIN {X -83.0014,Y 91.6486,Z 139,A 127.8978,B 24.2322,C -1.5497,E1 24.1724,E2 678.5775} C_DIS
LIN {X -79.75,Y 94.4921,Z 139,A 125.8481,B 24.2322,C -1.5522,E1 24.1768,E2 680.6294} C_DIS
LIN {X -76.2919,Y 97.305,Z 139,A 123.8408,B 24.2317,C -1.5592,E1 24.1811,E2 682.6273} C_DIS
LIN {X -73.1272,Y 99.7052,Z 139,A 122.0366,B 24.2313,C -1.5646,E1 24.1851,E2 684.4249} C_DIS
LIN {X -69.8272,Y 102.0435,Z 139,A 120.0852,B 24.2313,C -1.5651,E1 24.1896,E2 686.3821} C_DIS
LIN {X -66.2619,Y 104.3942,Z 139,A 118.4094,B 24.2303,C -1.5821,E1 24.1935,E2 688.0221} C_DIS
LIN {X -62.1414,Y 106.8981,Z 139,A 115.8883,B 24.2308,C -1.5737,E1 24.1996,E2 690.5716} C_DIS
LIN {X -58.8134,Y 108.7648,Z 139,A 114.0318,B 24.2308,C -1.5729,E1 24.2041,E2 692.4355} C_DIS
LIN {X -54.9794,Y 110.7501,Z 139,A 111.6449,B 24.2317,C -1.5594,E1 24.2102,E2 694.8619} C_DIS
LIN {X -51.1416,Y 112.5757,Z 139,A 110.0861,B 24.2304,C -1.5803,E1 24.214,E2 696.3738} C_DIS
LIN {X -47.6443,Y 114.0976,Z 139,A 108.4851,B 24.2298,C -1.5902,E1 24.2181,E2 697.9544} C_DIS
LIN {X -44.9021,Y 115.2045,Z 139,A 107.1053,B 24.2297,C -1.5916,E1 24.2217,E2 699.3338} C_DIS
LIN {X -42.4812,Y 116.1204,Z 139,A 105.5943,B 24.2304,C -1.5795,E1 24.2257,E2 700.8777} C_DIS
LIN {X -38.0409,Y 117.6492,Z 139,A 103.5828,B 24.2298,C -1.5893,E1 24.231,E2 702.8689} C_DIS
LIN {X -34.3073,Y 118.7918,Z 139,A 101.786,B 24.2297,C -1.5919,E1 24.2358,E2 704.6625} C_DIS
LIN {X -30.5107,Y 119.8223,Z 139,A 99.9861,B 24.2295,C -1.5948,E1 24.2406,E2 706.4583} C_DIS
LIN {X -27.8861,Y 120.4607,Z 139,A 98.711,B 24.2295,C -1.5948,E1 24.2441,E2 707.7348} C_DIS
LIN {X -23.8689,Y 121.322,Z 139,A 96.7633,B 24.2295,C -1.5945,E1 24.2494,E2 709.6858} C_DIS
LIN {X -20.3202,Y 121.9647,Z 139,A 95.1519,B 24.2293,C -1.5985,E1 24.2538,E2 711.2892} C_DIS
LIN {X -16.4183,Y 122.5516,Z 139,A 93.3084,B 24.2293,C -1.599,E1 24.2589,E2 713.133} C_DIS
LIN {X -12.8206,Y 122.9802,Z 139,A 91.596,B 24.2293,C -1.5984,E1 24.2637,E2 714.848} C_DIS
LIN {X -8.9969,Y 123.3183,Z 139,A 89.8588,B 24.2291,C -1.6011,E1 24.2685,E2 716.5795} C_DIS
LIN {X -5.1411,Y 123.5396,Z 139,A 88.0764,B 24.2291,C -1.602,E1 24.2735,E2 718.36} C_DIS
LIN {X -1.3565,Y 123.6405,Z 139,A 86.2317,B 24.2293,C -1.5983,E1 24.2787,E2 720.2138} C_DIS
LIN {X 2.5927,Y 123.6201,Z 139,A 84.3956,B 24.2293,C -1.5983,E1 24.2838,E2 722.0497} C_DIS
LIN {X 6.4811,Y 123.4764,Z 139,A 82.5818,B 24.2293,C -1.5979,E1 24.2888,E2 723.8638} C_DIS
LIN {X 10.5928,Y 123.1916,Z 139,A 80.8022,B 24.2289,C -1.6038,E1 24.2938,E2 725.6284} C_DIS
LIN {X 14.1611,Y 122.8333,Z 139,A 79.0575,B 24.2292,C -1.5997,E1 24.2986,E2 727.3817} C_DIS
LIN {X 17.9506,Y 122.3369,Z 139,A 77.3152,B 24.2292,C -1.6005,E1 24.3034,E2 729.1204} C_DIS
LIN {X 21.6255,Y 121.7402,Z 139,A 75.5894,B 24.2292,C -1.5999,E1 24.3082,E2 730.8458} C_DIS
LIN {X 28.2119,Y 120.3863,Z 139,A 72.4961,B 24.2292,C -1.5994,E1 24.3166,E2 733.9364} C_DIS
LIN {X 32.457,Y 119.3113,Z 139,A 70.4017,B 24.2295,C -1.5951,E1 24.3223,E2 736.0379} C_DIS
LIN {X 35.9814,Y 118.2948,Z 139,A 68.7975,B 24.2293,C -1.5983,E1 24.3266,E2 737.6315} C_DIS
LIN {X 39.337,Y 117.2218,Z 139,A 67.1615,B 24.2293,C -1.5967,E1 24.3309,E2 739.2679} C_DIS
LIN {X 43.1788,Y 115.8615,Z 139,A 65.2801,B 24.2295,C -1.5953,E1 24.3358,E2 741.1488} C_DIS
LIN {X 46.7614,Y 114.4637,Z 139,A 63.3874,B 24.2299,C -1.5883,E1 24.3408,E2 743.0541} C_DIS
LIN {X 50.3462,Y 112.9315,Z 139,A 61.8566,B 24.2292,C -1.5992,E1 24.3446,E2 744.5547} C_DIS
LIN {X 53.2594,Y 111.5871,Z 139,A 60.2826,B 24.2296,C -1.5933,E1 24.3486,E2 746.1389} C_DIS
LIN {X 55.9326,Y 110.2715,Z 139,A 58.8596,B 24.2298,C -1.5895,E1 24.3522,E2 747.567} C_DIS
LIN {X 58.6797,Y 108.8367,Z 139,A 57.4502,B 24.2298,C -1.5888,E1 24.3557,E2 748.974} C_DIS
LIN {X 62.0753,Y 106.9363,Z 139,A 55.6088,B 24.2301,C -1.5844,E1 24.3602,E2 750.8205} C_DIS
LIN {X 65.5653,Y 104.8331,Z 139,A 53.8431,B 24.23,C -1.5873,E1 24.3643,E2 752.5734} C_DIS
LIN {X 68.7448,Y 102.7758,Z 139,A 52.0543,B 24.2302,C -1.5828,E1 24.3685,E2 754.3669} C_DIS
LIN {X 71.2742,Y 101.038,Z 139,A 50.5614,B 24.2306,C -1.577,E1 24.372,E2 755.8686} C_DIS
LIN {X 74.1774,Y 98.927,Z 139,A 48.7759,B 24.2311,C -1.5683,E1 24.376,E2 757.6688} C_DIS
LIN {X 78.0976,Y 95.8618,Z 139,A 46.4508,B 24.2314,C -1.563,E1 24.3811,E2 759.9976} C_DIS
LIN {X 81.5669,Y 92.9282,Z 139,A 44.398,B 24.2315,C -1.5614,E1 24.3854,E2 762.0462} C_DIS
LIN {X 84.7313,Y 90.0518,Z 139,A 42.4506,B 24.2317,C -1.5589,E1 24.3894,E2 763.9913} C_DIS
LIN {X 87.9172,Y 86.9445,Z 139,A 40.4292,B 24.2318,C -1.5564,E1 24.3934,E2 766.01} C_DIS
LIN {X 90.6938,Y 84.0442,Z 139,A 38.5261,B 24.2322,C -1.5502,E1 24.3971,E2 767.9195} C_DIS
LIN {X 93.5303,Y 80.8754,Z 139,A 36.574,B 24.2324,C -1.5465,E1 24.4007,E2 769.8715} C_DIS
LIN {X 96.4372,Y 77.3864,Z 139,A 34.4861,B 24.2327,C -1.5423,E1 24.4044,E2 771.9598} C_DIS
LIN {X 99.0167,Y 74.0571,Z 139,A 32.2687,B 24.2337,C -1.5247,E1 24.4082,E2 774.209} C_DIS
LIN {X 101.0717,Y 71.2264,Z 139,A 31.0588,B 24.2328,C -1.5404,E1 24.4101,E2 775.3747} C_DIS
LIN {X 103.0548,Y 68.3268,Z 139,A 29.2816,B 24.2335,C -1.5289,E1 24.4129,E2 777.1706} C_DIS
LIN {X 105.4519,Y 64.5646,Z 139,A 27.2485,B 24.2337,C -1.525,E1 24.4159,E2 779.2024} C_DIS
LIN {X 107.668,Y 60.7977,Z 139,A 25.2778,B 24.2339,C -1.5222,E1 24.4186,E2 781.1695} C_DIS
LIN {X 109.4107,Y 57.5981,Z 139,A 23.7077,B 24.2339,C -1.5233,E1 24.4207,E2 782.7284} C_DIS
LIN {X 110.921,Y 54.6331,Z 139,A 21.8746,B 24.2349,C -1.5047,E1 24.423,E2 784.5963} C_DIS
LIN {X 112.948,Y 50.3093,Z 139,A 19.925,B 24.2345,C -1.5112,E1 24.4252,E2 786.5194} C_DIS
LIN {X 114.5107,Y 46.645,Z 139,A 18.0975,B 24.2348,C -1.5067,E1 24.4272,E2 788.3474} C_DIS
LIN {X 115.743,Y 43.4951,Z 139,A 16.6908,B 24.2346,C -1.5099,E1 24.4286,E2 789.7382} C_DIS
LIN {X 116.7622,Y 40.6803,Z 139,A 15.1507,B 24.2353,C -1.4982,E1 24.4301,E2 791.2977} C_DIS
LIN {X 119.0972,Y 33.2285,Z 139,A 11.5653,B 24.2358,C -1.4887,E1 24.433,E2 794.885} C_DIS
LIN {X 119.9968,Y 29.8233,Z 139,A 9.479,B 24.2374,C -1.4614,E1 24.4345,E2 797.0249} C_DIS
LIN {X 120.8735,Y 26.0363,Z 139,A 8.09,B 24.2366,C -1.4759,E1 24.4353,E2 798.3704} C_DIS
LIN {X 121.6601,Y 22.0732,Z 139,A 6.2801,B 24.2367,C -1.4731,E1 24.4362,E2 800.1764} C_DIS
LIN {X 122.2356,Y 18.6245,Z 139,A 4.5989,B 24.2372,C -1.4649,E1 24.4369,E2 801.8671} C_DIS
LIN {X 122.799,Y 14.4489,Z 139,A 2.6996,B 24.2374,C -1.4612,E1 24.4376,E2 803.7636} C_DIS
LIN {X 123.2204,Y 10.2524,Z 139,A 0.7551,B 24.2377,C -1.4554,E1 24.4381,E2 805.7104} C_DIS
LIN {X 123.4881,Y 6.2483,Z 139,A -1.0609,B 24.238,C -1.4515,E1 24.4384,E2 807.5246} C_DIS
LIN {X 123.6288,Y 2.0712,Z 139,A -2.9904,B 24.2383,C -1.4456,E1 24.4385,E2 809.4567} C_DIS
LIN {X 123.6331,Y -1.8144,Z 139,A -4.7777,B 24.2386,C -1.4404,E1 24.4385,E2 811.2456} C_DIS
LIN {X 123.5039,Y -5.9346,Z 139,A -6.6681,B 24.2389,C -1.4351,E1 24.4383,E2 813.1371} C_DIS
LIN {X 123.2792,Y -9.5318,Z 139,A -8.3189,B 24.2391,C -1.4306,E1 24.438,E2 814.7888} C_DIS
LIN {X 122.9379,Y -13.2139,Z 139,A -10.0029,B 24.2394,C -1.4265,E1 24.4375,E2 816.4724} C_DIS
LIN {X 122.4604,Y -17.0862,Z 139,A -11.8366,B 24.2398,C -1.4193,E1 24.4369,E2 818.3124} C_DIS
LIN {X 121.9301,Y -20.528,Z 139,A -13.4343,B 24.24,C -1.4148,E1 24.4362,E2 819.9112} C_DIS
LIN {X 120.7178,Y -26.7574,Z 139,A -16.4253,B 24.2407,C -1.4028,E1 24.4345,E2 822.9133} C_DIS
LIN {X 119.8729,Y -30.3114,Z 139,A -18.0236,B 24.2407,C -1.402,E1 24.4334,E2 824.5039} C_DIS
LIN {X 118.937,Y -33.8014,Z 139,A -19.9213,B 24.2416,C -1.3856,E1 24.432,E2 826.43} C_DIS
LIN {X 117.455,Y -38.6366,Z 139,A -21.8239,B 24.2408,C -1.3999,E1 24.4304,E2 828.2867} C_DIS
LIN {X 116.4407,Y -41.5928,Z 139,A -23.4895,B 24.2416,C -1.3846,E1 24.4289,E2 829.9798} C_DIS
LIN {X 115.3153,Y -44.6168,Z 139,A -24.9384,B 24.2418,C -1.3822,E1 24.4274,E2 831.4261} C_DIS
LIN {X 114.2233,Y -47.3433,Z 139,A -27.0564,B 24.2439,C -1.3409,E1 24.4251,E2 833.6321} C_DIS
LIN {X 111.9798,Y -52.4315,Z 139,A -28.9216,B 24.2425,C -1.3678,E1 24.423,E2 835.4217} C_DIS
LIN {X 110.2577,Y -55.9598,Z 139,A -30.3576,B 24.2418,C -1.3813,E1 24.4212,E2 836.8172} C_DIS
LIN {X 108.6944,Y -58.9433,Z 139,A -32.2314,B 24.2429,C -1.3611,E1 24.4187,E2 838.7297} C_DIS
LIN {X 106.8894,Y -62.1562,Z 139,A -33.9139,B 24.2431,C -1.3573,E1 24.4164,E2 840.4123} C_DIS
LIN {X 104.7946,Y -65.6271,Z 139,A -35.8689,B 24.2436,C -1.3481,E1 24.4135,E2 842.3793} C_DIS
LIN {X 102.4045,Y -69.2966,Z 139,A -37.7729,B 24.2436,C -1.3485,E1 24.4106,E2 844.2726} C_DIS
LIN {X 100.3689,Y -72.2143,Z 139,A -39.4075,B 24.2438,C -1.3446,E1 24.408,E2 845.9085} C_DIS
LIN {X 98.4694,Y -74.7838,Z 139,A -40.8606,B 24.2438,C -1.3419,E1 24.4055,E2 847.3609} C_DIS
LIN {X 95.6948,Y -78.302,Z 139,A -43.0194,B 24.2444,C -1.3323,E1 24.4018,E2 849.5326} C_DIS
LIN {X 92.8791,Y -81.6229,Z 139,A -45.0727,B 24.2448,C -1.3252,E1 24.398,E2 851.5933} C_DIS
LIN {X 90.8221,Y -83.9055,Z 139,A -46.4538,B 24.2448,C -1.3237,E1 24.3954,E2 852.9719} C_DIS
LIN {X 87.4177,Y -87.447,Z 139,A -48.754,B 24.2452,C -1.3169,E1 24.3909,E2 855.2785} C_DIS
LIN {X 84.1613,Y -90.5847,Z 139,A -50.7698,B 24.2452,C -1.3157,E1 24.3868,E2 857.2886} C_DIS
LIN {X 81.7179,Y -92.7951,Z 139,A -52.2779,B 24.2454,C -1.313,E1 24.3837,E2 858.7969} C_DIS
LIN {X 78.5279,Y -95.5102,Z 139,A -54.2709,B 24.2457,C -1.3061,E1 24.3794,E2 860.7987} C_DIS
LIN {X 75.2601,Y -98.1053,Z 139,A -56.1471,B 24.2458,C -1.3047,E1 24.3753,E2 862.6713} C_DIS
LIN {X 72.2904,Y -100.3141,Z 139,A -57.9139,B 24.2461,C -1.2986,E1 24.3713,E2 864.4464} C_DIS
LIN {X 68.2885,Y -103.0801,Z 139,A -60.1512,B 24.2463,C -1.2948,E1 24.3661,E2 866.685} C_DIS
LIN {X 64.4963,Y -105.4939,Z 139,A -62.1937,B 24.2464,C -1.2928,E1 24.3613,E2 868.7257} C_DIS
LIN {X 61.1355,Y -107.4763,Z 139,A -63.9128,B 24.2464,C -1.2937,E1 24.3571,E2 870.437} C_DIS
LIN {X 57.9795,Y -109.2104,Z 139,A -65.6376,B 24.2466,C -1.2881,E1 24.3529,E2 872.1703} C_DIS
LIN {X 54.9108,Y -110.7839,Z 139,A -67.1291,B 24.2466,C -1.2906,E1 24.3492,E2 873.6517} C_DIS
LIN {X 51.8219,Y -112.2619,Z 139,A -68.7248,B 24.2466,C -1.2876,E1 24.3451,E2 875.2503} C_DIS
LIN {X 48.7642,Y -113.624,Z 139,A -70.2827,B 24.2468,C -1.285,E1 24.3411,E2 876.8109} C_DIS
LIN {X 45.545,Y -114.9541,Z 139,A -72.0327,B 24.2472,C -1.2761,E1 24.3366,E2 878.5781} C_DIS
LIN {X 41.1328,Y -116.6053,Z 139,A -74.1406,B 24.2472,C -1.2768,E1 24.331,E2 880.6799} C_DIS
LIN {X 32.4033,Y -119.3257,Z 139,A -78.2767,B 24.2472,C -1.2766,E1 24.32,E2 884.8088} C_DIS
LIN {X 25.7661,Y -120.9319,Z 139,A -81.575,B 24.2477,C -1.2672,E1 24.311,E2 888.1251} C_DIS
LIN {X 21.649,Y -121.736,Z 139,A -83.4368,B 24.2476,C -1.2695,E1 24.3059,E2 889.9793} C_DIS
LIN {X 17.5555,Y -122.3933,Z 139,A -85.339,B 24.2476,C -1.269,E1 24.3007,E2 891.8808} C_DIS
LIN {X 13.4913,Y -122.908,Z 139,A -87.2728,B 24.2477,C -1.2662,E1 24.2953,E2 893.82} C_DIS
LIN {X 9.7198,Y -123.2653,Z 139,A -89.0935,B 24.2479,C -1.2622,E1 24.2902,E2 895.6492} C_DIS
LIN {X 5.9446,Y -123.5034,Z 139,A -90.7976,B 24.2479,C -1.2638,E1 24.2855,E2 897.3489} C_DIS
LIN {X 1.9662,Y -123.6305,Z 139,A -92.6035,B 24.2478,C -1.2651,E1 24.2804,E2 899.1514} C_DIS
LIN {X 1.9662,Y -123.6305,Z 139,A -92.6035,B 24.2478,C -1.2651,E1 24.2804,E2 899.1514} C_DIS
Enddeposition()
LIN {X 0.8753,Y -122.6632,Z 139,A -92.5938,B 23.6838,C -1.1932,E1 23.7135,E2 899.2418} C_DIS
Startdeposition()
$VEL.CP = VEL_PRINT
LIN {X 3.3494,Y -122.6214,Z 139,A -91.0451,B 23.6829,C -1.2114,E1 23.7179,E2 897.6482} C_DIS
LIN {X 7.1186,Y -122.4611,Z 139,A -89.4684,B 23.6833,C -1.2036,E1 23.7223,E2 896.0915} C_DIS
LIN {X 10.5238,Y -122.2149,Z 139,A -87.745,B 23.683,C -1.2102,E1 23.7271,E2 894.3525} C_DIS
LIN {X 14.2042,Y -121.8422,Z 139,A -86.0064,B 23.683,C -1.2117,E1 23.732,E2 892.6115} C_DIS
LIN {X 17.539,Y -121.4067,Z 139,A -84.3545,B 23.6827,C -1.2164,E1 23.7366,E2 890.9492} C_DIS
LIN {X 20.9719,Y -120.8626,Z 139,A -82.8133,B 23.6827,C -1.2138,E1 23.7408,E2 889.4162} C_DIS
LIN {X 23.9276,Y -120.3118,Z 139,A -81.2518,B 23.6824,C -1.2223,E1 23.7451,E2 887.8357} C_DIS
LIN {X 27.6944,Y -119.5003,Z 139,A -79.4821,B 23.6824,C -1.2226,E1 23.7499,E2 886.0677} C_DIS
LIN {X 32.041,Y -118.4091,Z 139,A -77.3838,B 23.6823,C -1.225,E1 23.7556,E2 883.9669} C_DIS
LIN {X 36.2342,Y -117.1936,Z 139,A -75.333,B 23.6821,C -1.2278,E1 23.7611,E2 881.9129} C_DIS
LIN {X 39.9001,Y -115.9965,Z 139,A -73.553,B 23.6821,C -1.2291,E1 23.7658,E2 880.1334} C_DIS
LIN {X 44.147,Y -114.4476,Z 139,A -71.4582,B 23.682,C -1.2311,E1 23.7713,E2 878.0383} C_DIS
LIN {X 48.3238,Y -112.7477,Z 139,A -69.5048,B 23.6822,C -1.227,E1 23.7763,E2 876.0998} C_DIS
LIN {X 51.0718,Y -111.5301,Z 139,A -67.9418,B 23.6817,C -1.2367,E1 23.7803,E2 874.5171} C_DIS
LIN {X 55.0377,Y -109.6285,Z 139,A -66.0108,B 23.6818,C -1.2342,E1 23.7851,E2 872.5977} C_DIS
LIN {X 57.8323,Y -108.1806,Z 139,A -64.4536,B 23.6815,C -1.2408,E1 23.789,E2 871.0288} C_DIS
LIN {X 61.7692,Y -105.9823,Z 139,A -62.3222,B 23.6812,C -1.2458,E1 23.7942,E2 868.8918} C_DIS
LIN {X 65.6252,Y -103.6384,Z 139,A -60.2466,B 23.6812,C -1.2483,E1 23.7991,E2 866.817} C_DIS
LIN {X 69.3839,Y -101.1603,Z 139,A -58.2964,B 23.6812,C -1.2452,E1 23.8036,E2 864.8813} C_DIS
LIN {X 72.5153,Y -98.9399,Z 139,A -56.3785,B 23.6808,C -1.2549,E1 23.808,E2 862.9466} C_DIS
LIN {X 76.056,Y -96.2453,Z 139,A -54.284,B 23.6805,C -1.2601,E1 23.8126,E2 860.8473} C_DIS
LIN {X 79.2307,Y -93.6489,Z 139,A -52.4429,B 23.6805,C -1.2609,E1 23.8165,E2 859.0119} C_DIS
LIN {X 82.1224,Y -91.124,Z 139,A -50.594,B 23.6801,C -1.2677,E1 23.8204,E2 857.1539} C_DIS
LIN {X 85.1217,Y -88.3285,Z 139,A -48.7025,B 23.68,C -1.2711,E1 23.8242,E2 855.2621} C_DIS
LIN {X 88.306,Y -85.145,Z 139,A -46.6292,B 23.6798,C -1.2749,E1 23.8283,E2 853.1889} C_DIS
LIN {X 91.1246,Y -82.1218,Z 139,A -44.6707,B 23.6795,C -1.2811,E1 23.832,E2 851.224} C_DIS
LIN {X 94.0775,Y -78.721,Z 139,A -42.673,B 23.6795,C -1.2815,E1 23.8356,E2 849.2351} C_DIS
LIN {X 96.6905,Y -75.4892,Z 139,A -40.6609,B 23.679,C -1.2901,E1 23.8391,E2 847.2116} C_DIS
LIN {X 98.9403,Y -72.5147,Z 139,A -38.9186,B 23.6787,C -1.2949,E1 23.842,E2 845.4663} C_DIS
LIN {X 101.5366,Y -68.8323,Z 139,A -36.8262,B 23.6785,C -1.3002,E1 23.8453,E2 843.3717} C_DIS
LIN {X 103.9683,Y -65.1019,Z 139,A -34.9126,B 23.6785,C -1.2981,E1 23.8482,E2 841.4737} C_DIS
LIN {X 105.9813,Y -61.771,Z 139,A -32.9571,B 23.678,C -1.31,E1 23.851,E2 839.4992} C_DIS
LIN {X 108.1796,Y -57.8342,Z 139,A -30.8519,B 23.6776,C -1.3162,E1 23.8538,E2 837.3905} C_DIS
LIN {X 109.8771,Y -54.5362,Z 139,A -29.2895,B 23.6778,C -1.3132,E1 23.8558,E2 835.8444} C_DIS
LIN {X 111.4963,Y -51.1449,Z 139,A -27.4433,B 23.6773,C -1.3229,E1 23.858,E2 833.9847} C_DIS
LIN {X 113.0642,Y -47.5783,Z 139,A -25.6156,B 23.677,C -1.3288,E1 23.86,E2 832.1529} C_DIS
LIN {X 114.696,Y -43.4992,Z 139,A -23.7234,B 23.677,C -1.3274,E1 23.8619,E2 830.2753} C_DIS
LIN {X 116.0002,Y -39.8893,Z 139,A -21.9427,B 23.6768,C -1.3325,E1 23.8636,E2 828.4928} C_DIS
LIN {X 116.9387,Y -37.0478,Z 139,A -20.5517,B 23.6766,C -1.3365,E1 23.8648,E2 827.1} C_DIS
LIN {X 117.8156,Y -34.1574,Z 139,A -19.0181,B 23.676,C -1.347,E1 23.866,E2 825.55} C_DIS
LIN {X 118.9897,Y -29.8117,Z 139,A -16.9225,B 23.6757,C -1.3533,E1 23.8675,E2 823.4513} C_DIS
LIN {X 119.9768,Y -25.5508,Z 139,A -15.0294,B 23.6757,C -1.3526,E1 23.8686,E2 821.5716} C_DIS
LIN {X 120.7102,Y -21.8232,Z 139,A -13.2084,B 23.6753,C -1.3606,E1 23.8696,E2 819.7422} C_DIS
LIN {X 121.2875,Y -18.3492,Z 139,A -11.5817,B 23.675,C -1.365,E1 23.8703,E2 818.1147} C_DIS
LIN {X 121.746,Y -15.011,Z 139,A -9.9198,B 23.6745,C -1.3744,E1 23.8709,E2 816.4401} C_DIS
LIN {X 122.1543,Y -11.2154,Z 139,A -8.3302,B 23.6747,C -1.3708,E1 23.8713,E2 814.8693} C_DIS
LIN {X 122.4235,Y -7.7278,Z 139,A -6.6349,B 23.6743,C -1.3791,E1 23.8716,E2 813.1642} C_DIS
LIN {X 122.5899,Y -4.3704,Z 139,A -5.0019,B 23.6738,C -1.3873,E1 23.8718,E2 811.5213} C_DIS
LIN {X 122.6678,Y -0.2798,Z 139,A -3.1768,B 23.6738,C -1.3893,E1 23.8718,E2 809.7027} C_DIS
LIN {X 122.6116,Y 3.7007,Z 139,A -1.2772,B 23.6733,C -1.3973,E1 23.8718,E2 807.7954} C_DIS
LIN {X 122.4359,Y 7.5263,Z 139,A 0.3921,B 23.6733,C -1.3973,E1 23.8715,E2 806.1366} C_DIS
LIN {X 122.2147,Y 10.5267,Z 139,A 1.7814,B 23.6731,C -1.401,E1 23.8712,E2 804.7467} C_DIS
LIN {X 121.8418,Y 14.2083,Z 139,A 3.5106,B 23.6727,C -1.4066,E1 23.8707,E2 803.0146} C_DIS
LIN {X 121.419,Y 17.4531,Z 139,A 5.0749,B 23.6724,C -1.4132,E1 23.8701,E2 801.4437} C_DIS
LIN {X 120.862,Y 20.975,Z 139,A 6.6852,B 23.6722,C -1.4158,E1 23.8694,E2 799.8371} C_DIS
LIN {X 120.1705,Y 24.6216,Z 139,A 8.4351,B 23.6719,C -1.422,E1 23.8684,E2 798.0826} C_DIS
LIN {X 119.3453,Y 28.3549,Z 139,A 10.3201,B 23.6713,C -1.4324,E1 23.8672,E2 796.1836} C_DIS
LIN {X 118.4095,Y 32.0394,Z 139,A 12.0868,B 23.671,C -1.4374,E1 23.866,E2 794.4152} C_DIS
LIN {X 117.1924,Y 36.2379,Z 139,A 13.9604,B 23.6711,C -1.4355,E1 23.8645,E2 792.5576} C_DIS
LIN {X 116.0126,Y 39.8537,Z 139,A 15.8948,B 23.6704,C -1.4485,E1 23.8627,E2 790.6027} C_DIS
LIN {X 114.4486,Y 44.1444,Z 139,A 17.9884,B 23.6701,C -1.4529,E1 23.8607,E2 788.5105} C_DIS
LIN {X 112.757,Y 48.3024,Z 139,A 19.9367,B 23.6701,C -1.4519,E1 23.8586,E2 786.5761} C_DIS
LIN {X 111.5252,Y 51.0825,Z 139,A 21.3409,B 23.67,C -1.4552,E1 23.857,E2 785.1718} C_DIS
LIN {X 110.2334,Y 53.8139,Z 139,A 22.7361,B 23.6698,C -1.4584,E1 23.8553,E2 783.7766} C_DIS
LIN {X 108.8827,Y 56.4978,Z 139,A 24.112,B 23.6696,C -1.461,E1 23.8536,E2 782.4019} C_DIS
LIN {X 107.1318,Y 59.7534,Z 139,A 26.0236,B 23.6688,C -1.4746,E1 23.851,E2 780.4674} C_DIS
LIN {X 104.7995,Y 63.7551,Z 139,A 28.1573,B 23.6686,C -1.479,E1 23.8479,E2 778.3344} C_DIS
LIN {X 102.4436,Y 67.4749,Z 139,A 30.1638,B 23.6684,C -1.482,E1 23.8449,E2 776.3312} C_DIS
LIN {X 100.2994,Y 70.6228,Z 139,A 31.9743,B 23.668,C -1.488,E1 23.842,E2 774.5151} C_DIS
LIN {X 98.0432,Y 73.7233,Z 139,A 33.7334,B 23.6679,C -1.491,E1 23.8391,E2 772.7577} C_DIS
LIN {X 95.3041,Y 77.2318,Z 139,A 35.7559,B 23.6677,C -1.4933,E1 23.8356,E2 770.7395} C_DIS
LIN {X 92.6595,Y 80.3859,Z 139,A 37.748,B 23.6673,C -1.5011,E1 23.8319,E2 768.7377} C_DIS
LIN {X 89.6364,Y 83.7431,Z 139,A 39.7589,B 23.6673,C -1.5011,E1 23.8282,E2 766.7359} C_DIS
LIN {X 86.741,Y 86.7393,Z 139,A 41.7817,B 23.6668,C -1.509,E1 23.8242,E2 764.7029} C_DIS
LIN {X 83.7416,Y 89.6377,Z 139,A 43.6892,B 23.6667,C -1.5112,E1 23.8203,E2 762.7984} C_DIS
LIN {X 80.3926,Y 92.6536,Z 139,A 45.8053,B 23.6664,C -1.5159,E1 23.8159,E2 760.6794} C_DIS
LIN {X 77.2303,Y 95.3053,Z 139,A 47.7201,B 23.6662,C -1.519,E1 23.8117,E2 758.7648} C_DIS
LIN {X 73.7215,Y 98.0445,Z 139,A 49.6505,B 23.6664,C -1.5159,E1 23.8075,E2 756.8497} C_DIS
LIN {X 70.6373,Y 100.2892,Z 139,A 51.5623,B 23.6658,C -1.525,E1 23.8031,E2 754.9223} C_DIS
LIN {X 66.924,Y 102.8044,Z 139,A 53.6643,B 23.6656,C -1.5288,E1 23.7982,E2 752.8184} C_DIS
LIN {X 63.0679,Y 105.2145,Z 139,A 55.6139,B 23.6659,C -1.5239,E1 23.7936,E2 750.8873} C_DIS
LIN {X 60.4318,Y 106.7506,Z 139,A 57.1872,B 23.6654,C -1.5328,E1 23.7898,E2 749.2968} C_DIS
LIN {X 56.6364,Y 108.8099,Z 139,A 59.0693,B 23.6656,C -1.5294,E1 23.7852,E2 747.4289} C_DIS
LIN {X 53.8118,Y 110.2345,Z 139,A 60.6781,B 23.6651,C -1.5373,E1 23.7811,E2 745.8051} C_DIS
LIN {X 50.4704,Y 111.8034,Z 139,A 62.3104,B 23.6652,C -1.5351,E1 23.777,E2 744.1826} C_DIS
LIN {X 47.4628,Y 113.1124,Z 139,A 63.9002,B 23.6649,C -1.5395,E1 23.7729,E2 742.586} C_DIS
LIN {X 43.4925,Y 114.6986,Z 139,A 65.7622,B 23.6652,C -1.5353,E1 23.7681,E2 740.7388} C_DIS
LIN {X 40.5617,Y 115.7671,Z 139,A 67.3592,B 23.6647,C -1.543,E1 23.7638,E2 739.1261} C_DIS
LIN {X 37.051,Y 116.9377,Z 139,A 68.943,B 23.665,C -1.5378,E1 23.7597,E2 737.5583} C_DIS
LIN {X 34.167,Y 117.8128,Z 139,A 70.4791,B 23.6646,C -1.5447,E1 23.7555,E2 736.0079} C_DIS
LIN {X 29.8036,Y 118.9917,Z 139,A 72.6014,B 23.6646,C -1.5465,E1 23.7498,E2 733.8845} C_DIS
LIN {X 26.1055,Y 119.857,Z 139,A 74.3535,B 23.6646,C -1.5465,E1 23.745,E2 732.135} C_DIS
LIN {X 22.4534,Y 120.5958,Z 139,A 75.9581,B 23.6648,C -1.5411,E1 23.7407,E2 730.5458} C_DIS
LIN {X 19.4917,Y 121.1104,Z 139,A 77.499,B 23.6644,C -1.5477,E1 23.7364,E2 728.9901} C_DIS
LIN {X 15.8029,Y 121.6448,Z 139,A 79.1212,B 23.6647,C -1.5429,E1 23.7319,E2 727.3814} C_DIS
LIN {X 12.0241,Y 122.0766,Z 139,A 80.8938,B 23.6647,C -1.543,E1 23.727,E2 725.6098} C_DIS
LIN {X 8.2245,Y 122.3929,Z 139,A 82.8176,B 23.6643,C -1.5495,E1 23.7216,E2 723.671} C_DIS
LIN {X 4.5165,Y 122.5842,Z 139,A 84.5487,B 23.6643,C -1.5493,E1 23.7168,E2 721.9409} C_DIS
LIN {X 0.6942,Y 122.6652,Z 139,A 86.1643,B 23.6648,C -1.5415,E1 23.7123,E2 720.3449} C_DIS
LIN {X -2.3126,Y 122.6456,Z 139,A 87.7407,B 23.6644,C -1.5488,E1 23.7079,E2 718.7503} C_DIS
LIN {X -6.6335,Y 122.4885,Z 139,A 89.7318,B 23.6644,C -1.5468,E1 23.7023,E2 716.7635} C_DIS
LIN {X -9.8364,Y 122.273,Z 139,A 91.0898,B 23.6649,C -1.54,E1 23.6986,E2 715.422} C_DIS
LIN {X -13.5192,Y 121.9204,Z 139,A 92.8492,B 23.6649,C -1.5405,E1 23.6937,E2 713.6603} C_DIS
LIN {X -17.1908,Y 121.4565,Z 139,A 94.6052,B 23.6649,C -1.5406,E1 23.6888,E2 711.9026} C_DIS
LIN {X -20.2748,Y 120.9798,Z 139,A 96.106,B 23.6649,C -1.5415,E1 23.6847,E2 710.3981} C_DIS
LIN {X -23.9601,Y 120.3051,Z 139,A 97.9559,B 23.6646,C -1.5445,E1 23.6796,E2 708.5386} C_DIS
LIN {X -27.6857,Y 119.5023,Z 139,A 99.7194,B 23.6648,C -1.5422,E1 23.6748,E2 706.7785} C_DIS
LIN {X -32.0519,Y 118.4062,Z 139,A 101.8379,B 23.6648,C -1.5408,E1 23.6691,E2 704.6602} C_DIS
LIN {X -36.2658,Y 117.1839,Z 139,A 103.7349,B 23.6654,C -1.5319,E1 23.6641,E2 702.7819} C_DIS
LIN {X -39.2299,Y 116.2256,Z 139,A 105.3568,B 23.6651,C -1.5374,E1 23.6597,E2 701.1432} C_DIS
LIN {X -42.7754,Y 114.9672,Z 139,A 107.0037,B 23.6655,C -1.5304,E1 23.6554,E2 699.5103} C_DIS
LIN {X -46.1928,Y 113.6374,Z 139,A 108.8442,B 23.6653,C -1.5335,E1 23.6506,E2 697.6575} C_DIS
LIN {X -50.4315,Y 111.8209,Z 139,A 110.9842,B 23.6655,C -1.5298,E1 23.6452,E2 695.5215} C_DIS
LIN {X -53.8133,Y 110.2337,Z 139,A 112.5802,B 23.6661,C -1.5206,E1 23.6412,E2 693.944} C_DIS
LIN {X -56.5019,Y 108.8805,Z 139,A 114.1067,B 23.6659,C -1.5235,E1 23.6374,E2 692.406} C_DIS
LIN {X -59.7426,Y 107.1378,Z 139,A 115.7283,B 23.6664,C -1.5164,E1 23.6334,E2 690.7973} C_DIS
LIN {X -62.3403,Y 105.647,Z 139,A 117.1474,B 23.6664,C -1.5147,E1 23.63,E2 689.3777} C_DIS
LIN {X -65.5928,Y 103.6588,Z 139,A 119.0362,B 23.6664,C -1.516,E1 23.6255,E2 687.4794} C_DIS
LIN {X -68.8322,Y 101.5366,Z 139,A 120.8792,B 23.6664,C -1.5139,E1 23.6212,E2 685.6352} C_DIS
LIN {X -72.5144,Y 98.9405,Z 139,A 122.9868,B 23.6667,C -1.5098,E1 23.6164,E2 683.5301} C_DIS
LIN {X -76.0577,Y 96.244,Z 139,A 125.1039,B 23.6669,C -1.5069,E1 23.6118,E2 681.412} C_DIS
Enddeposition()
END
